C07284=1031.312,-76.674,415.942,167.658,41.793,157.756
C07285=1031.305,-76.924,415.953,167.656,41.794,157.756
C07286=1031.300,-77.174,415.964,167.653,41.796,157.756
C07287=1031.294,-77.423,415.975,167.650,41.797,157.756
C07288=1031.287,-77.673,415.985,167.647,41.798,157.757
C07289=1031.281,-77.922,415.996,167.644,41.799,157.757
C07290=1031.275,-78.172,416.007,167.642,41.801,157.757
C07291=1031.269,-78.422,416.018,167.639,41.802,157.757
C07292=1031.263,-78.672,416.029,167.636,41.803,157.757
C07293=1031.258,-78.921,416.040,167.633,41.805,157.757
C07294=1031.251,-79.171,416.051,167.630,41.806,157.757
C07295=1031.246,-79.421,416.062,167.628,41.808,157.757
C07296=1031.239,-79.670,416.073,167.625,41.809,157.757
C07297=1031.233,-79.920,416.084,167.622,41.811,157.757
C07298=1031.227,-80.170,416.094,167.619,41.812,157.757
C07299=1031.222,-80.420,416.105,167.617,41.814,157.757
C07300=1031.214,-80.670,416.116,167.614,41.815,157.757
C07301=1031.209,-80.919,416.126,167.611,41.816,157.757
C07302=1031.202,-81.168,416.137,167.608,41.818,157.758
C07303=1031.196,-81.418,416.148,167.606,41.820,157.758
C07304=1031.190,-81.669,416.158,167.603,41.821,157.758
C07305=1031.184,-81.918,416.168,167.600,41.823,157.758
C07306=1031.178,-82.167,416.179,167.597,41.825,157.758
C07307=1031.171,-82.417,416.190,167.594,41.826,157.758
C07308=1031.165,-82.667,416.201,167.592,41.827,157.758
C07309=1031.160,-82.917,416.211,167.589,41.828,157.758
C07310=1031.153,-83.166,416.221,167.586,41.830,157.758
C07311=1031.147,-83.416,416.233,167.582,41.832,157.758
C07312=1031.141,-83.666,416.243,167.580,41.833,157.758
C07313=1031.135,-83.915,416.253,167.577,41.835,157.759
C07314=1031.128,-84.199,416.266,167.574,41.837,157.759
C07315=1031.121,-84.485,416.278,167.570,41.839,157.759
C07316=1031.114,-84.769,416.290,167.568,41.840,157.759
C07317=1031.107,-85.054,416.302,167.564,41.842,157.759
C07318=1031.101,-85.303,416.312,167.561,41.843,157.759
C07319=1031.096,-85.553,416.322,167.558,41.845,157.759
C07320=1031.089,-85.803,416.333,167.556,41.847,157.759
C07321=1031.083,-86.053,416.344,167.553,41.848,157.759
C07322=1031.077,-86.303,416.354,167.550,41.850,157.760
C07323=1031.071,-86.552,416.364,167.547,41.851,157.760
C07324=1031.065,-86.802,416.374,167.545,41.852,157.760
C07325=1031.059,-87.051,416.385,167.542,41.854,157.760
C07326=1031.053,-87.302,416.396,167.539,41.855,157.760
C07327=1031.046,-87.551,416.405,167.536,41.857,157.760
C07328=1031.041,-87.801,416.416,167.534,41.859,157.760
C07329=1031.035,-88.050,416.427,167.531,41.860,157.760
C07330=1031.029,-88.300,416.437,167.528,41.862,157.760
C07331=1031.023,-88.550,416.448,167.525,41.863,157.760
C07332=1031.017,-88.799,416.457,167.522,41.865,157.760
C07333=1031.010,-89.050,416.468,167.520,41.866,157.761
C07334=1031.004,-89.299,416.478,167.517,41.868,157.761
C07335=1030.999,-89.549,416.489,167.514,41.869,157.761
C07336=1030.992,-89.798,416.499,167.510,41.871,157.761
C07337=1030.987,-90.048,416.509,167.508,41.873,157.761
C07338=1030.981,-90.298,416.520,167.505,41.874,157.761
C07339=1030.975,-90.547,416.530,167.502,41.876,157.761
C07340=1030.969,-90.797,416.541,167.499,41.877,157.761
C07341=1030.963,-91.047,416.550,167.496,41.878,157.761
C07342=1030.957,-91.296,416.561,167.494,41.880,157.761
C07343=1030.951,-91.546,416.571,167.491,41.882,157.761
C07344=1030.945,-91.796,416.582,167.488,41.883,157.761
C07345=1030.938,-92.046,416.591,167.485,41.885,157.762
C07346=1030.933,-92.296,416.602,167.483,41.887,157.762
C07347=1030.926,-92.545,416.612,167.480,41.888,157.762
C07348=1030.921,-92.795,416.622,167.477,41.889,157.762
C07349=1030.915,-93.045,416.632,167.475,41.891,157.762
C07350=1030.909,-93.295,416.643,167.472,41.892,157.762
C07351=1030.903,-93.544,416.653,167.469,41.894,157.762
C07352=1030.897,-93.794,416.663,167.466,41.895,157.762
C07353=1030.892,-94.044,416.673,167.463,41.897,157.762
C07354=1030.885,-94.293,416.683,167.460,41.899,157.762
C07355=1030.880,-94.543,416.694,167.457,41.900,157.762
C07356=1030.873,-94.793,416.704,167.454,41.902,157.763
C07357=1030.868,-95.043,416.714,167.451,41.903,157.763
C07358=1030.862,-95.292,416.724,167.448,41.904,157.763
C07359=1030.856,-95.542,416.734,167.446,41.906,157.763
C07360=1030.850,-95.792,416.744,167.443,41.908,157.763
C07361=1030.844,-96.042,416.754,167.440,41.909,157.763
C07362=1030.839,-96.290,416.764,167.437,41.911,157.763
C07363=1030.833,-96.540,416.774,167.435,41.913,157.763
C07364=1030.827,-96.790,416.784,167.432,41.914,157.763
C07365=1030.821,-97.040,416.795,167.429,41.915,157.763
C07366=1030.815,-97.290,416.804,167.426,41.917,157.764
C07367=1030.810,-97.540,416.814,167.424,41.918,157.764
C07368=1030.803,-97.789,416.824,167.421,41.920,157.764
C07369=1030.797,-98.039,416.834,167.417,41.922,157.764
C07370=1030.792,-98.289,416.844,167.414,41.924,157.764
C07371=1030.785,-98.539,416.854,167.412,41.925,157.764
C07372=1030.779,-98.788,416.864,167.409,41.927,157.764
C07373=1030.773,-99.038,416.873,167.406,41.929,157.764
C07374=1030.768,-99.288,416.883,167.404,41.930,157.764
C07375=1030.761,-99.538,416.893,167.401,41.932,157.764
C07376=1030.755,-99.787,416.903,167.398,41.934,157.765
C07377=1030.749,-100.037,416.913,167.394,41.936,157.765
C07378=1030.743,-100.324,416.924,167.392,41.937,157.765
C07379=1030.736,-100.611,416.935,167.388,41.939,157.765
C07380=1030.729,-100.898,416.946,167.385,41.941,157.765
C07381=1030.722,-101.184,416.957,167.382,41.943,157.765
C07382=1030.716,-101.434,416.967,167.379,41.945,157.765
C07383=1030.710,-101.684,416.977,167.376,41.946,157.765
C07384=1030.704,-101.934,416.986,167.373,41.948,157.766
C07385=1030.698,-102.184,416.996,167.371,41.950,157.766
C07386=1030.693,-102.433,417.005,167.367,41.952,157.766
C07387=1030.686,-102.683,417.015,167.364,41.954,157.766
C07388=1030.681,-102.933,417.025,167.361,41.955,157.766
C07389=1030.674,-103.182,417.035,167.359,41.956,157.766
C07390=1030.668,-103.432,417.045,167.356,41.958,157.766
C07391=1030.662,-103.682,417.054,167.353,41.960,157.766
C07392=1030.657,-103.931,417.063,167.351,41.962,157.766
C07393=1030.651,-104.182,417.073,167.348,41.964,157.767
C07394=1030.645,-104.431,417.083,167.344,41.965,157.767
C07395=1030.639,-104.681,417.092,167.341,41.967,157.767
C07396=1030.633,-104.931,417.102,167.339,41.968,157.767
C07397=1030.627,-105.180,417.111,167.336,41.970,157.767
C07398=1030.622,-105.430,417.121,167.333,41.972,157.767
C07399=1030.616,-105.680,417.131,167.330,41.974,157.767
C07400=1030.610,-105.930,417.140,167.328,41.975,157.767
C07401=1030.603,-106.180,417.150,167.325,41.977,157.767
C07402=1030.598,-106.429,417.159,167.321,41.979,157.768
C07403=1030.592,-106.678,417.169,167.319,41.981,157.768
C07404=1030.586,-106.929,417.179,167.316,41.983,157.768
C07405=1030.580,-107.179,417.188,167.313,41.984,157.768
C07406=1030.575,-107.428,417.197,167.310,41.985,157.768
C07407=1030.569,-107.678,417.206,167.308,41.987,157.768
C07408=1030.562,-107.928,417.216,167.305,41.989,157.768
C07409=1030.556,-108.177,417.225,167.301,41.991,157.768
C07410=1030.551,-108.427,417.235,167.299,41.993,157.768
C07411=1030.545,-108.677,417.244,167.296,41.995,157.769
C07412=1030.539,-108.927,417.253,167.293,41.996,157.769
C07413=1030.533,-109.176,417.262,167.290,41.998,157.769
C07414=1030.527,-109.426,417.272,167.288,42.000,157.769
C07415=1030.521,-109.676,417.281,167.284,42.002,157.769
C07416=1030.515,-109.926,417.290,167.281,42.004,157.769
C07417=1030.509,-110.175,417.300,167.279,42.005,157.769
C07418=1030.503,-110.425,417.309,167.276,42.008,157.770
C07419=1030.497,-110.675,417.318,167.273,42.010,157.770
C07420=1030.492,-110.924,417.327,167.270,42.011,157.770
C07421=1030.486,-111.174,417.337,167.267,42.013,157.770
C07422=1030.480,-111.425,417.346,167.264,42.015,157.770
C07423=1030.474,-111.674,417.355,167.262,42.017,157.770
C07424=1030.468,-111.923,417.364,167.259,42.019,157.770
C07425=1030.462,-112.174,417.373,167.256,42.020,157.770
C07426=1030.457,-112.423,417.382,167.252,42.022,157.771
C07427=1030.450,-112.673,417.392,167.250,42.024,157.771
C07428=1030.444,-112.923,417.401,167.247,42.026,157.771
C07429=1030.439,-113.172,417.410,167.244,42.028,157.771
C07430=1030.433,-113.422,417.420,167.242,42.029,157.771
C07431=1030.427,-113.672,417.428,167.239,42.031,157.771
C07432=1030.421,-113.922,417.438,167.235,42.033,157.771
C07433=1030.415,-114.172,417.446,167.233,42.035,157.771
C07434=1030.410,-114.421,417.456,167.230,42.037,157.772
C07435=1030.404,-114.671,417.465,167.227,42.038,157.772
C07436=1030.398,-114.920,417.473,167.224,42.040,157.772
C07437=1030.392,-115.170,417.483,167.222,42.042,157.772
C07438=1030.386,-115.420,417.492,167.218,42.044,157.772
C07439=1030.380,-115.670,417.501,167.215,42.046,157.772
C07440=1030.374,-115.920,417.510,167.213,42.047,157.772
C07441=1030.369,-116.169,417.519,167.210,42.050,157.772
C07442=1030.361,-116.456,417.528,167.206,42.052,157.773
C07443=1030.355,-116.743,417.539,167.203,42.054,157.773
C07444=1030.348,-117.028,417.549,167.200,42.056,157.773
C07445=1030.342,-117.315,417.559,167.196,42.058,157.773
C07446=1030.336,-117.565,417.568,167.194,42.060,157.773
C07447=1030.330,-117.815,417.577,167.191,42.062,157.773
C07448=1030.325,-118.064,417.587,167.188,42.064,157.774
C07449=1030.318,-118.314,417.595,167.185,42.066,157.774
C07450=1030.312,-118.563,417.604,167.182,42.068,157.774
C07451=1030.306,-118.814,417.613,167.179,42.070,157.774
C07452=1030.301,-119.064,417.622,167.177,42.071,157.774
C07453=1030.294,-119.313,417.630,167.174,42.073,157.774
C07454=1030.288,-119.563,417.639,167.170,42.075,157.774
C07455=1030.283,-119.813,417.648,167.168,42.078,157.774
C07456=1030.277,-120.063,417.657,167.165,42.079,157.775
C07457=1030.272,-120.313,417.666,167.162,42.081,157.775
C07458=1030.265,-120.561,417.674,167.159,42.083,157.775
C07459=1030.260,-120.812,417.683,167.156,42.085,157.775
C07460=1030.254,-121.061,417.692,167.153,42.087,157.775
C07461=1030.248,-121.312,417.700,167.151,42.089,157.775
C07462=1030.242,-121.561,417.709,167.148,42.091,157.775
C07463=1030.236,-121.811,417.718,167.144,42.093,157.776
C07464=1030.231,-122.061,417.726,167.142,42.095,157.776
C07465=1030.225,-122.311,417.736,167.139,42.096,157.776
C07466=1030.219,-122.560,417.744,167.136,42.099,157.776
C07467=1030.213,-122.810,417.753,167.134,42.101,157.776
C07468=1030.208,-123.060,417.761,167.130,42.103,157.776
C07469=1030.202,-123.309,417.770,167.127,42.104,157.776
C07470=1030.196,-123.559,417.779,167.124,42.106,157.777
C07471=1030.190,-123.809,417.787,167.122,42.108,157.777
C07472=1030.184,-124.059,417.796,167.119,42.110,157.777
C07473=1030.179,-124.309,417.804,167.116,42.112,157.777
C07474=1030.173,-124.558,417.813,167.113,42.114,157.777
C07475=1030.167,-124.808,417.822,167.110,42.116,157.777
C07476=1030.161,-125.058,417.830,167.108,42.118,157.777
C07477=1030.155,-125.308,417.839,167.104,42.120,157.778
C07478=1030.150,-125.558,417.847,167.101,42.122,157.778
C07479=1030.144,-125.807,417.855,167.098,42.124,157.778
C07480=1030.138,-126.058,417.864,167.096,42.126,157.778
C07481=1030.132,-126.307,417.872,167.092,42.128,157.778
C07482=1030.126,-126.556,417.881,167.090,42.130,157.778
C07483=1030.121,-126.807,417.890,167.087,42.133,157.779
C07484=1030.115,-127.056,417.898,167.084,42.134,157.779
C07485=1030.109,-127.306,417.907,167.082,42.136,157.779
C07486=1030.103,-127.556,417.914,167.078,42.139,157.779
C07487=1030.097,-127.806,417.923,167.075,42.140,157.779
C07488=1030.092,-128.055,417.932,167.073,42.142,157.779
C07489=1030.087,-128.305,417.941,167.070,42.143,157.779
C07490=1030.082,-128.554,417.951,167.067,42.144,157.779
C07491=1030.080,-128.803,417.962,167.065,42.145,157.779
C07492=1030.076,-129.053,417.973,167.063,42.144,157.779
C07493=1030.074,-129.303,417.984,167.059,42.144,157.779
C07494=1030.072,-129.554,417.996,167.058,42.143,157.778
C07495=1030.071,-129.803,418.009,167.056,42.142,157.778
C07496=1030.071,-130.053,418.022,167.053,42.139,157.777
C07497=1030.071,-130.303,418.036,167.051,42.137,157.777
C07498=1030.071,-130.553,418.050,167.049,42.134,157.776
C07499=1030.073,-130.803,418.066,167.048,42.131,157.776
C07500=1030.075,-131.053,418.082,167.045,42.127,157.775
C07501=1030.077,-131.302,418.098,167.044,42.123,157.774
C07502=1030.081,-131.553,418.115,167.043,42.118,157.773
C07503=1030.085,-131.803,418.132,167.042,42.112,157.772
C07504=1030.089,-132.053,418.150,167.040,42.107,157.771
C07505=1030.095,-132.302,418.169,167.039,42.101,157.770
C07506=1029.776,-132.327,417.864,166.990,42.343,157.807
C07507=1029.771,-132.078,417.846,166.992,42.349,157.808
C07508=1029.767,-131.828,417.828,166.993,42.355,157.809
C07509=1029.762,-131.577,417.810,166.994,42.360,157.811
C07510=1029.759,-131.327,417.794,166.996,42.365,157.811
C07511=1029.756,-131.077,417.777,166.997,42.369,157.812
C07512=1029.755,-130.827,417.762,166.999,42.373,157.813
C07513=1029.753,-130.578,417.747,167.001,42.376,157.814
C07514=1029.752,-130.328,417.732,167.003,42.379,157.814
C07515=1029.752,-130.078,417.718,167.004,42.382,157.815
C07516=1029.753,-129.828,417.705,167.007,42.383,157.815
C07517=1029.754,-129.578,417.692,167.009,42.385,157.816
C07518=1029.755,-129.328,417.680,167.011,42.386,157.816
C07519=1029.758,-129.079,417.668,167.013,42.387,157.816
C07520=1029.760,-128.829,417.657,167.016,42.386,157.816
C07521=1029.764,-128.579,417.646,167.018,42.386,157.816
C07522=1029.769,-128.330,417.636,167.021,42.386,157.817
C07523=1029.773,-128.080,417.627,167.024,42.384,157.816
C07524=1029.778,-127.830,417.619,167.027,42.382,157.816
C07525=1029.784,-127.580,417.610,167.029,42.380,157.816
C07526=1029.790,-127.332,417.602,167.032,42.378,157.816
C07527=1029.795,-127.082,417.593,167.036,42.376,157.816
C07528=1029.802,-126.832,417.585,167.038,42.374,157.816
C07529=1029.807,-126.582,417.576,167.041,42.372,157.816
C07530=1029.812,-126.332,417.568,167.044,42.370,157.816
C07531=1029.819,-126.082,417.560,167.047,42.368,157.815
C07532=1029.824,-125.833,417.551,167.050,42.366,157.815
C07533=1029.830,-125.583,417.543,167.053,42.364,157.815
C07534=1029.836,-125.333,417.534,167.055,42.362,157.815
C07535=1029.841,-125.083,417.526,167.059,42.360,157.815
C07536=1029.848,-124.833,417.518,167.062,42.358,157.815
C07537=1029.854,-124.584,417.508,167.064,42.355,157.814
C07538=1029.860,-124.334,417.501,167.068,42.353,157.814
C07539=1029.865,-124.084,417.492,167.070,42.352,157.814
C07540=1029.871,-123.834,417.483,167.073,42.349,157.814
C07541=1029.877,-123.584,417.474,167.076,42.347,157.814
C07542=1029.883,-123.335,417.466,167.078,42.345,157.814
C07543=1029.888,-123.085,417.457,167.082,42.344,157.814
C07544=1029.894,-122.835,417.448,167.085,42.342,157.813
C07545=1029.900,-122.586,417.441,167.087,42.339,157.813
C07546=1029.906,-122.335,417.432,167.090,42.337,157.813
C07547=1029.911,-122.086,417.422,167.094,42.335,157.813
C07548=1029.917,-121.836,417.414,167.096,42.334,157.813
C07549=1029.923,-121.586,417.406,167.099,42.331,157.813
C07550=1029.929,-121.337,417.397,167.102,42.329,157.813
C07551=1029.935,-121.087,417.388,167.105,42.327,157.812
C07552=1029.940,-120.837,417.379,167.108,42.326,157.812
C07553=1029.947,-120.587,417.371,167.110,42.323,157.812
C07554=1029.952,-120.338,417.362,167.113,42.321,157.812
C07555=1029.958,-120.087,417.353,167.116,42.320,157.812
C07556=1029.963,-119.838,417.344,167.120,42.318,157.812
C07557=1029.970,-119.588,417.335,167.122,42.316,157.812
C07558=1029.976,-119.338,417.327,167.125,42.313,157.811
C07559=1029.981,-119.088,417.318,167.127,42.311,157.811
C07560=1029.987,-118.839,417.309,167.131,42.310,157.811
C07561=1029.993,-118.589,417.300,167.134,42.308,157.811
C07562=1029.998,-118.339,417.291,167.137,42.306,157.811
C07563=1030.005,-118.089,417.283,167.139,42.303,157.811
C07564=1030.010,-117.840,417.274,167.143,42.302,157.811
C07565=1030.016,-117.590,417.265,167.145,42.300,157.810
C07566=1030.022,-117.340,417.256,167.148,42.298,157.810
C07567=1030.029,-117.054,417.246,167.152,42.295,157.810
C07568=1030.035,-116.768,417.235,167.154,42.293,157.810
C07569=1030.042,-116.481,417.226,167.158,42.292,157.810
C07570=1030.049,-116.195,417.215,167.162,42.289,157.810
C07571=1030.055,-115.945,417.206,167.164,42.287,157.810
C07572=1030.061,-115.695,417.197,167.167,42.285,157.809
C07573=1030.066,-115.446,417.188,167.170,42.284,157.809
C07574=1030.073,-115.196,417.179,167.173,42.281,157.809
C07575=1030.078,-114.947,417.170,167.176,42.279,157.809
C07576=1030.084,-114.696,417.161,167.179,42.277,157.809
C07577=1030.090,-114.446,417.152,167.181,42.275,157.809
C07578=1030.096,-114.197,417.143,167.185,42.274,157.809
C07579=1030.102,-113.947,417.134,167.188,42.272,157.809
C07580=1030.107,-113.697,417.125,167.190,42.270,157.808
C07581=1030.113,-113.447,417.116,167.193,42.268,157.808
C07582=1030.119,-113.198,417.106,167.196,42.266,157.808
C07583=1030.125,-112.948,417.098,167.199,42.265,157.808
C07584=1030.131,-112.698,417.088,167.202,42.263,157.808
C07585=1030.136,-112.448,417.080,167.205,42.260,157.808
C07586=1030.142,-112.199,417.070,167.207,42.258,157.808
C07587=1030.148,-111.949,417.060,167.210,42.257,157.807
C07588=1030.154,-111.699,417.052,167.213,42.255,157.807
C07589=1030.160,-111.449,417.042,167.217,42.253,157.807
C07590=1030.166,-111.199,417.033,167.219,42.251,157.807
C07591=1030.171,-110.950,417.024,167.222,42.249,157.807
C07592=1030.177,-110.700,417.015,167.225,42.247,157.807
C07593=1030.184,-110.450,417.005,167.227,42.246,157.807
C07594=1030.189,-110.200,416.997,167.231,42.244,157.807
C07595=1030.195,-109.951,416.987,167.234,42.242,157.807
C07596=1030.201,-109.701,416.978,167.236,42.240,157.806
C07597=1030.207,-109.452,416.968,167.239,42.238,157.806
C07598=1030.213,-109.201,416.959,167.242,42.237,157.806
C07599=1030.219,-108.951,416.950,167.246,42.235,157.806
C07600=1030.224,-108.702,416.941,167.248,42.233,157.806
C07601=1030.231,-108.453,416.931,167.251,42.230,157.806
C07602=1030.236,-108.202,416.922,167.253,42.229,157.806
C07603=1030.243,-107.952,416.913,167.256,42.227,157.805
C07604=1030.248,-107.703,416.904,167.260,42.225,157.805
C07605=1030.254,-107.453,416.894,167.263,42.223,157.805
C07606=1030.261,-107.204,416.884,167.265,42.221,157.805
C07607=1030.266,-106.953,416.876,167.268,42.219,157.805
C07608=1030.272,-106.704,416.866,167.271,42.218,157.805
C07609=1030.278,-106.454,416.857,167.273,42.216,157.805
C07610=1030.284,-106.204,416.847,167.277,42.214,157.805
C07611=1030.290,-105.954,416.837,167.280,42.213,157.805
C07612=1030.295,-105.705,416.828,167.283,42.211,157.804
C07613=1030.302,-105.456,416.818,167.285,42.209,157.804
C07614=1030.308,-105.206,416.809,167.288,42.207,157.804
C07615=1030.314,-104.956,416.799,167.291,42.206,157.804
C07616=1030.319,-104.705,416.790,167.294,42.204,157.804
C07617=1030.325,-104.456,416.780,167.297,42.202,157.804
C07618=1030.331,-104.206,416.771,167.300,42.200,157.804
C07619=1030.337,-103.957,416.761,167.302,42.198,157.804
C07620=1030.343,-103.707,416.752,167.305,42.197,157.803
C07621=1030.348,-103.457,416.742,167.308,42.195,157.803
C07622=1030.354,-103.208,416.732,167.311,42.193,157.803
C07623=1030.360,-102.958,416.723,167.314,42.191,157.803
C07624=1030.366,-102.708,416.713,167.317,42.189,157.803
C07625=1030.373,-102.458,416.704,167.320,42.188,157.803
C07626=1030.378,-102.208,416.694,167.323,42.186,157.803
C07627=1030.384,-101.959,416.684,167.325,42.185,157.803
C07628=1030.390,-101.709,416.675,167.328,42.183,157.803
C07629=1030.396,-101.459,416.665,167.332,42.181,157.803
C07630=1030.402,-101.210,416.654,167.334,42.179,157.802
C07631=1030.408,-100.923,416.643,167.337,42.177,157.802
C07632=1030.416,-100.636,416.632,167.341,42.175,157.802
C07633=1030.422,-100.349,416.621,167.344,42.173,157.802
C07634=1030.429,-100.063,416.610,167.347,42.171,157.802
C07635=1030.435,-99.813,416.601,167.350,42.169,157.802
C07636=1030.441,-99.563,416.591,167.352,42.167,157.802
C07637=1030.447,-99.313,416.581,167.356,42.165,157.802
C07638=1030.453,-99.063,416.572,167.359,42.164,157.802
C07639=1030.460,-98.814,416.561,167.362,42.163,157.801
C07640=1030.465,-98.564,416.551,167.364,42.161,157.801
C07641=1030.471,-98.314,416.542,167.367,42.159,157.801
C07642=1030.477,-98.064,416.532,167.370,42.157,157.801
C07643=1030.483,-97.815,416.522,167.373,42.155,157.801
C07644=1030.489,-97.564,416.512,167.376,42.154,157.801
C07645=1030.495,-97.315,416.502,167.379,42.152,157.801
C07646=1030.501,-97.065,416.492,167.382,42.151,157.801
C07647=1030.506,-96.816,416.483,167.384,42.149,157.800
C07648=1030.512,-96.566,416.473,167.387,42.147,157.800
C07649=1030.518,-96.317,416.462,167.390,42.146,157.800
C07650=1030.524,-96.067,416.452,167.393,42.144,157.800
C07651=1030.530,-95.817,416.443,167.395,42.142,157.800
C07652=1030.536,-95.567,416.432,167.398,42.141,157.800
C07653=1030.542,-95.318,416.422,167.401,42.140,157.800
C07654=1030.547,-95.067,416.412,167.405,42.138,157.800
C07655=1030.554,-94.818,416.402,167.407,42.136,157.800
C07656=1030.559,-94.568,416.391,167.410,42.134,157.800
C07657=1030.565,-94.318,416.382,167.413,42.133,157.800
C07658=1030.571,-94.069,416.371,167.416,42.131,157.799
C07659=1030.577,-93.819,416.361,167.418,42.129,157.799
C07660=1030.583,-93.570,416.351,167.421,42.128,157.799
C07661=1030.589,-93.320,416.341,167.424,42.127,157.799
C07662=1030.595,-93.070,416.331,167.427,42.125,157.799
C07663=1030.601,-92.821,416.321,167.429,42.123,157.799
C07664=1030.607,-92.570,416.310,167.432,42.122,157.799
C07665=1030.612,-92.321,416.300,167.436,42.120,157.799
C07666=1030.618,-92.071,416.290,167.439,42.118,157.799
C07667=1030.624,-91.822,416.279,167.441,42.117,157.799
C07668=1030.630,-91.572,416.270,167.444,42.115,157.799
C07669=1030.636,-91.322,416.259,167.447,42.113,157.798
C07670=1030.642,-91.073,416.249,167.449,42.112,157.798
C07671=1030.648,-90.822,416.239,167.452,42.111,157.798
C07672=1030.654,-90.573,416.229,167.455,42.109,157.798
C07673=1030.660,-90.322,416.218,167.458,42.107,157.798
C07674=1030.667,-90.073,416.208,167.461,42.106,157.798
C07675=1030.672,-89.823,416.198,167.463,42.104,157.798
C07676=1030.679,-89.574,416.187,167.466,42.102,157.798
C07677=1030.684,-89.324,416.176,167.470,42.100,157.798
C07678=1030.690,-89.074,416.166,167.473,42.099,157.798
C07679=1030.696,-88.825,416.156,167.475,42.098,157.798
C07680=1030.702,-88.575,416.146,167.478,42.096,157.797
C07681=1030.708,-88.326,416.136,167.481,42.095,157.797
C07682=1030.714,-88.076,416.125,167.484,42.093,157.797
C07683=1030.721,-87.826,416.115,167.486,42.091,157.797
C07684=1030.726,-87.576,416.104,167.489,42.089,157.797
C07685=1030.732,-87.326,416.094,167.492,42.088,157.797
C07686=1030.738,-87.077,416.083,167.495,42.087,157.797
C07687=1030.744,-86.827,416.073,167.497,42.085,157.797
C07688=1030.750,-86.578,416.063,167.500,42.084,157.797
C07689=1030.757,-86.328,416.052,167.503,42.082,157.797
C07690=1030.763,-86.078,416.042,167.507,42.080,157.797
C07691=1030.768,-85.828,416.031,167.509,42.079,157.797
C07692=1030.774,-85.579,416.020,167.512,42.077,157.796
C07693=1030.780,-85.329,416.011,167.515,42.075,157.796
C07694=1030.786,-85.080,416.000,167.517,42.074,157.796
C07695=1030.793,-84.794,415.988,167.520,42.072,157.796
C07696=1030.801,-84.510,415.976,167.524,42.070,157.796
C07697=1030.808,-84.225,415.964,167.527,42.069,157.796
C07698=1030.814,-83.941,415.953,167.530,42.067,157.796
C07699=1030.820,-83.691,415.942,167.533,42.065,157.796
C07700=1030.827,-83.442,415.931,167.536,42.063,157.796
C07701=1030.833,-83.192,415.920,167.539,42.062,157.795
C07702=1030.838,-82.942,415.910,167.541,42.060,157.795
C07703=1030.845,-82.692,415.900,167.544,42.059,157.795
C07704=1030.851,-82.443,415.889,167.547,42.057,157.795
C07705=1030.858,-82.193,415.878,167.550,42.056,157.795
C07706=1030.863,-81.943,415.868,167.552,42.054,157.795
C07707=1030.869,-81.694,415.857,167.556,42.052,157.795
C07708=1030.876,-81.444,415.846,167.559,42.050,157.795
C07709=1030.882,-81.194,415.836,167.562,42.049,157.795
C07710=1030.888,-80.945,415.825,167.564,42.047,157.795
C07711=1030.894,-80.695,415.815,167.567,42.046,157.794
C07712=1030.900,-80.445,415.804,167.570,42.045,157.794
C07713=1030.906,-80.195,415.794,167.573,42.043,157.794
C07714=1030.912,-79.946,415.783,167.575,42.041,157.794
C07715=1030.918,-79.696,415.771,167.578,42.040,157.794
C07716=1030.924,-79.446,415.761,167.581,42.038,157.794
C07717=1030.931,-79.197,415.750,167.584,42.037,157.794
C07718=1030.937,-78.947,415.739,167.586,42.035,157.794
C07719=1030.943,-78.697,415.728,167.589,42.034,157.794
C07720=1030.948,-78.448,415.717,167.592,42.032,157.794
C07721=1030.955,-78.198,415.706,167.595,42.031,157.794
C07722=1030.961,-77.948,415.695,167.598,42.030,157.794
C07723=1030.966,-77.699,415.684,167.600,42.028,157.793
C07724=1030.973,-77.449,415.673,167.603,42.027,157.793
C07725=1030.979,-77.199,415.663,167.606,42.025,157.793
C07726=1030.985,-76.950,415.652,167.609,42.024,157.793
C07727=1030.991,-76.700,415.641,167.611,42.022,157.793
C07728=1030.997,-76.450,415.630,167.614,42.021,157.793
C07729=1031.003,-76.201,415.619,167.617,42.019,157.793
C07730=1031.009,-75.951,415.608,167.620,42.018,157.793
C07731=1031.015,-75.701,415.597,167.623,42.016,157.793
C07732=1031.020,-75.452,415.586,167.625,42.015,157.793
C07733=1031.028,-75.202,415.575,167.628,42.014,157.793
C07734=1031.033,-74.952,415.564,167.631,42.012,157.793
C07735=1031.040,-74.702,415.553,167.634,42.011,157.793
C07736=1031.045,-74.453,415.542,167.637,42.010,157.793
C07737=1031.051,-74.203,415.531,167.639,42.008,157.792
C07738=1031.058,-73.953,415.519,167.642,42.007,157.792
C07739=1031.064,-73.704,415.509,167.645,42.005,157.792
C07740=1031.070,-73.454,415.497,167.648,42.004,157.792
C07741=1031.075,-73.204,415.486,167.651,42.003,157.792
C07742=1031.081,-72.955,415.475,167.653,42.001,157.792
C07743=1031.087,-72.705,415.463,167.656,42.000,157.792
C07744=1031.093,-72.455,415.452,167.659,41.999,157.792
C07745=1031.099,-72.205,415.441,167.662,41.997,157.792
C07746=1031.105,-71.956,415.430,167.665,41.996,157.792
C07747=1031.110,-71.707,415.418,167.668,41.995,157.792
C07748=1031.117,-71.456,415.407,167.670,41.993,157.792
C07749=1031.122,-71.207,415.396,167.672,41.992,157.792
C07750=1031.129,-70.957,415.384,167.675,41.991,157.792
C07751=1031.135,-70.708,415.373,167.678,41.989,157.792
C07752=1031.141,-70.458,415.362,167.681,41.988,157.792
C07753=1031.146,-70.208,415.349,167.683,41.987,157.792
C07754=1031.153,-69.958,415.338,167.686,41.985,157.791
C07755=1031.159,-69.709,415.327,167.689,41.984,157.791
C07756=1031.165,-69.460,415.316,167.692,41.983,157.791
C07757=1031.171,-69.210,415.304,167.695,41.981,157.791
C07758=1031.176,-68.960,415.293,167.697,41.980,157.791
C07759=1031.183,-68.678,415.281,167.700,41.979,157.791
C07760=1031.190,-68.395,415.268,167.703,41.978,157.791
C07761=1031.197,-68.113,415.254,167.707,41.976,157.791
C07762=1031.204,-67.830,415.241,167.710,41.975,157.791
C07763=1031.210,-67.580,415.230,167.712,41.973,157.791
C07764=1031.216,-67.330,415.219,167.715,41.972,157.791
C07765=1031.222,-67.081,415.206,167.718,41.971,157.791
C07766=1031.228,-66.831,415.195,167.721,41.969,157.791
C07767=1031.234,-66.582,415.183,167.724,41.968,157.791
C07768=1031.240,-66.332,415.172,167.726,41.967,157.791
C07769=1031.247,-66.082,415.161,167.729,41.965,157.791
C07770=1031.252,-65.833,415.149,167.732,41.964,157.791
C07771=1031.258,-65.583,415.137,167.734,41.963,157.791
C07772=1031.265,-65.333,415.126,167.737,41.961,157.790
C07773=1031.271,-65.084,415.114,167.739,41.960,157.790
C07774=1031.277,-64.834,415.103,167.742,41.959,157.790
C07775=1031.282,-64.585,415.091,167.745,41.957,157.790
C07776=1031.289,-64.334,415.080,167.748,41.956,157.790
C07777=1031.295,-64.086,415.068,167.751,41.954,157.790
C07778=1031.301,-63.835,415.057,167.753,41.953,157.790
C07779=1031.307,-63.586,415.044,167.756,41.952,157.790
C07780=1031.313,-63.336,415.033,167.759,41.950,157.790
C07781=1031.319,-63.086,415.021,167.762,41.949,157.790
C07782=1031.326,-62.836,415.010,167.765,41.948,157.790
C07783=1031.331,-62.587,414.998,167.766,41.947,157.790
C07784=1031.338,-62.338,414.986,167.769,41.946,157.790
C07785=1031.343,-62.088,414.975,167.772,41.944,157.790
C07786=1031.350,-61.838,414.963,167.775,41.943,157.790
C07787=1031.356,-61.588,414.952,167.778,41.942,157.790
C07788=1031.362,-61.339,414.940,167.781,41.941,157.790
C07789=1031.368,-61.090,414.928,167.783,41.939,157.789
C07790=1031.375,-60.839,414.917,167.786,41.938,157.789
C07791=1031.381,-60.590,414.905,167.789,41.936,157.789
C07792=1031.387,-60.341,414.892,167.792,41.935,157.789
C07793=1031.393,-60.090,414.881,167.795,41.934,157.789
C07794=1031.399,-59.842,414.870,167.797,41.932,157.789
C07795=1031.406,-59.592,414.858,167.799,41.931,157.789
C07796=1031.411,-59.341,414.846,167.802,41.930,157.789
C07797=1031.418,-59.092,414.834,167.805,41.928,157.789
C07798=1031.424,-58.843,414.822,167.808,41.927,157.789
C07799=1031.430,-58.593,414.811,167.811,41.926,157.789
C07800=1031.436,-58.343,414.798,167.813,41.924,157.789
C07801=1031.443,-58.093,414.786,167.816,41.923,157.789
C07802=1031.449,-57.844,414.775,167.819,41.922,157.789
C07803=1031.455,-57.594,414.763,167.822,41.920,157.789
C07804=1031.461,-57.344,414.751,167.825,41.919,157.789
C07805=1031.468,-57.095,414.739,167.827,41.918,157.788
C07806=1031.474,-56.846,414.727,167.829,41.917,157.788
C07807=1031.480,-56.595,414.716,167.832,41.915,157.788
C07808=1031.486,-56.346,414.704,167.835,41.914,157.788
C07809=1031.493,-56.096,414.692,167.838,41.913,157.788
C07810=1031.499,-55.847,414.680,167.840,41.912,157.788
C07811=1031.505,-55.598,414.668,167.843,41.910,157.788
C07812=1031.511,-55.347,414.656,167.846,41.909,157.788
C07813=1031.518,-55.098,414.644,167.849,41.907,157.788
C07814=1031.524,-54.848,414.632,167.852,41.906,157.788
C07815=1031.530,-54.599,414.620,167.854,41.905,157.788
C07816=1031.536,-54.349,414.608,167.856,41.903,157.788
C07817=1031.543,-54.100,414.596,167.859,41.902,157.788
C07818=1031.549,-53.849,414.584,167.862,41.901,157.788
C07819=1031.555,-53.600,414.573,167.865,41.899,157.787
C07820=1031.562,-53.350,414.561,167.867,41.898,157.787
C07821=1031.567,-53.101,414.548,167.870,41.896,157.787
C07822=1031.574,-52.852,414.536,167.873,41.895,157.787
C07823=1031.581,-52.569,414.523,167.876,41.894,157.787
C07824=1031.588,-52.289,414.509,167.879,41.893,157.787
C07825=1031.595,-52.007,414.496,167.882,41.891,157.787
C07826=1031.603,-51.727,414.482,167.885,41.890,157.787
C07827=1031.609,-51.477,414.469,167.888,41.888,157.787
C07828=1031.615,-51.227,414.458,167.891,41.887,157.787
C07829=1031.622,-50.978,414.446,167.894,41.886,157.787
C07830=1031.628,-50.727,414.434,167.895,41.884,157.787
C07831=1031.634,-50.478,414.422,167.898,41.883,157.787
C07832=1031.640,-50.229,414.409,167.901,41.882,157.787
C07833=1031.647,-49.979,414.397,167.904,41.881,157.787
C07834=1031.653,-49.730,414.384,167.907,41.880,157.787
C07835=1031.658,-49.480,414.372,167.909,41.879,157.787
C07836=1031.664,-49.230,414.359,167.911,41.877,157.786
C07837=1031.671,-48.980,414.347,167.914,41.876,157.786
C07838=1031.677,-48.730,414.335,167.917,41.875,157.786
C07839=1031.683,-48.480,414.322,167.920,41.874,157.786
C07840=1031.689,-48.232,414.311,167.923,41.873,157.786
C07841=1031.695,-47.982,414.297,167.925,41.872,157.786
C07842=1031.701,-47.732,414.285,167.928,41.871,157.786
C07843=1031.708,-47.483,414.273,167.930,41.869,157.786
C07844=1031.714,-47.233,414.260,167.933,41.868,157.786
C07845=1031.719,-46.983,414.248,167.936,41.867,157.786
C07846=1031.726,-46.733,414.236,167.938,41.866,157.786
C07847=1031.732,-46.484,414.222,167.941,41.865,157.786
C07848=1031.738,-46.234,414.210,167.944,41.864,157.786
C07849=1031.745,-45.985,414.198,167.947,41.863,157.786
C07850=1031.751,-45.735,414.185,167.949,41.861,157.786
C07851=1031.757,-45.486,414.172,167.951,41.860,157.786
C07852=1031.764,-45.236,414.160,167.954,41.859,157.786
C07853=1031.770,-44.986,414.148,167.957,41.858,157.786
C07854=1031.775,-44.736,414.135,167.960,41.857,157.786
C07855=1031.782,-44.487,414.122,167.962,41.856,157.786
C07856=1031.788,-44.237,414.110,167.964,41.855,157.786
C07857=1031.794,-43.988,414.097,167.967,41.853,157.786
C07858=1031.800,-43.738,414.085,167.970,41.852,157.786
C07859=1031.807,-43.489,414.072,167.973,41.851,157.786
C07860=1031.813,-43.239,414.059,167.975,41.850,157.786
C07861=1031.819,-42.989,414.047,167.978,41.849,157.786
C07862=1031.826,-42.740,414.034,167.980,41.848,157.785
C07863=1031.832,-42.490,414.022,167.983,41.847,157.785
C07864=1031.838,-42.240,414.009,167.986,41.845,157.785
C07865=1031.844,-41.991,413.996,167.988,41.844,157.785
C07866=1031.851,-41.741,413.984,167.991,41.843,157.785
C07867=1031.857,-41.492,413.971,167.994,41.842,157.785
C07868=1031.863,-41.242,413.958,167.997,41.841,157.785
C07869=1031.869,-40.993,413.946,167.999,41.840,157.785
C07870=1031.876,-40.743,413.933,168.001,41.838,157.785
C07871=1031.881,-40.494,413.920,168.004,41.837,157.785
C07872=1031.887,-40.244,413.908,168.007,41.836,157.785
C07873=1031.894,-39.995,413.895,168.010,41.835,157.785
C07874=1031.900,-39.745,413.883,168.012,41.834,157.785
C07875=1031.906,-39.496,413.869,168.014,41.833,157.785
C07876=1031.912,-39.246,413.857,168.017,41.831,157.785
C07877=1031.919,-38.997,413.844,168.020,41.830,157.785
C07878=1031.926,-38.746,413.831,168.023,41.829,157.785
C07879=1031.932,-38.497,413.818,168.025,41.828,157.785
C07880=1031.938,-38.247,413.805,168.028,41.827,157.785
C07881=1031.944,-37.998,413.792,168.030,41.826,157.785
C07882=1031.950,-37.748,413.779,168.032,41.825,157.785
C07883=1031.956,-37.499,413.766,168.035,41.824,157.785
C07884=1031.962,-37.249,413.754,168.038,41.823,157.785
C07885=1031.968,-36.999,413.740,168.041,41.822,157.785
C07886=1031.975,-36.750,413.727,168.043,41.821,157.784
C07887=1031.982,-36.469,413.713,168.046,41.820,157.784
C07888=1031.989,-36.188,413.699,168.049,41.819,157.784
C07889=1031.995,-35.908,413.683,168.051,41.817,157.784
C07890=1032.002,-35.626,413.669,168.055,41.816,157.784
C07891=1032.009,-35.377,413.656,168.057,41.815,157.784
C07892=1032.015,-35.128,413.642,168.060,41.814,157.784
C07893=1032.021,-34.878,413.630,168.063,41.813,157.784
C07894=1032.027,-34.629,413.616,168.065,41.812,157.784
C07895=1032.034,-34.379,413.603,168.067,41.811,157.784
C07896=1032.040,-34.129,413.590,168.070,41.809,157.784
C07897=1032.046,-33.879,413.577,168.073,41.808,157.784
C07898=1032.052,-33.630,413.564,168.075,41.807,157.784
C07899=1032.058,-33.380,413.551,168.078,41.806,157.784
C07900=1032.064,-33.131,413.538,168.081,41.805,157.784
C07901=1032.071,-32.881,413.524,168.083,41.804,157.784
C07902=1032.077,-32.631,413.512,168.086,41.803,157.784
C07903=1032.083,-32.382,413.498,168.088,41.802,157.784
C07904=1032.089,-32.133,413.485,168.091,41.801,157.784
C07905=1032.096,-31.883,413.472,168.093,41.800,157.784
C07906=1032.102,-31.633,413.459,168.096,41.799,157.784
C07907=1032.108,-31.384,413.446,168.099,41.798,157.784
C07908=1032.115,-31.134,413.432,168.101,41.797,157.784
C07909=1032.121,-30.885,413.419,168.104,41.796,157.784
C07910=1032.127,-30.634,413.406,168.107,41.795,157.784
C07911=1032.133,-30.385,413.393,168.108,41.794,157.784
C07912=1032.140,-30.136,413.380,168.111,41.793,157.784
C07913=1032.146,-29.887,413.366,168.114,41.792,157.784
C07914=1032.153,-29.637,413.353,168.117,41.791,157.784
C07915=1032.159,-29.387,413.340,168.119,41.790,157.784
C07916=1032.165,-29.138,413.327,168.122,41.788,157.783
C07917=1032.171,-28.888,413.314,168.124,41.787,157.783
C07918=1032.178,-28.638,413.300,168.126,41.786,157.783
C07919=1032.184,-28.389,413.287,168.129,41.785,157.783
C07920=1032.190,-28.140,413.274,168.132,41.784,157.783
C07921=1032.197,-27.890,413.260,168.135,41.783,157.783
C07922=1032.203,-27.640,413.247,168.137,41.782,157.783
C07923=1032.209,-27.391,413.234,168.140,41.781,157.783
C07924=1032.215,-27.141,413.221,168.142,41.780,157.783
C07925=1032.221,-26.891,413.207,168.144,41.779,157.783
C07926=1032.228,-26.642,413.193,168.147,41.778,157.783
C07927=1032.234,-26.393,413.180,168.150,41.777,157.783
C07928=1032.240,-26.142,413.166,168.152,41.776,157.783
C07929=1032.246,-25.893,413.153,168.155,41.775,157.783
C07930=1032.252,-25.644,413.139,168.157,41.775,157.783
C07931=1032.259,-25.393,413.125,168.160,41.773,157.783
C07932=1032.265,-25.144,413.112,168.163,41.772,157.783
C07933=1032.271,-24.895,413.099,168.164,41.771,157.783
C07934=1032.277,-24.646,413.085,168.167,41.770,157.783
C07935=1032.283,-24.395,413.071,168.170,41.769,157.783
C07936=1032.289,-24.146,413.058,168.172,41.768,157.783
C07937=1032.296,-23.897,413.044,168.175,41.767,157.783
C07938=1032.302,-23.647,413.030,168.178,41.766,157.783
C07939=1032.308,-23.398,413.016,168.180,41.765,157.783
C07940=1032.314,-23.149,413.003,168.183,41.765,157.783
C07941=1032.321,-22.899,412.989,168.185,41.764,157.783
C07942=1032.327,-22.649,412.975,168.187,41.763,157.783
C07943=1032.334,-22.334,412.958,168.190,41.762,157.783
C07944=1032.343,-22.019,412.941,168.194,41.760,157.783
C07945=1032.351,-21.704,412.924,168.197,41.759,157.783
C07946=1032.359,-21.389,412.907,168.200,41.758,157.783
C07947=1032.364,-21.156,412.894,168.203,41.757,157.783
C07948=1032.370,-20.923,412.881,168.204,41.756,157.783
C07949=1032.376,-20.690,412.868,168.207,41.755,157.783
C07950=1032.382,-20.458,412.855,168.209,41.754,157.783
C07951=1032.388,-20.225,412.842,168.212,41.753,157.783
C07952=1032.394,-19.992,412.829,168.214,41.752,157.783
C07953=1032.400,-19.759,412.817,168.217,41.751,157.783
C07954=1032.405,-19.526,412.804,168.219,41.750,157.783
C07955=1032.412,-19.277,412.791,168.222,41.749,157.783
C07956=1032.418,-19.027,412.776,168.224,41.748,157.782
C07957=1032.424,-18.778,412.763,168.226,41.747,157.782
C07958=1032.431,-18.528,412.749,168.228,41.746,157.782
C07959=1032.436,-18.278,412.735,168.231,41.745,157.782
C07960=1032.443,-18.029,412.721,168.234,41.744,157.782
C07961=1032.450,-17.780,412.707,168.236,41.743,157.782
C07962=1032.455,-17.530,412.694,168.239,41.742,157.782
C07963=1032.462,-17.280,412.680,168.242,41.742,157.782
C07964=1032.469,-17.031,412.666,168.244,41.741,157.782
C07965=1032.475,-16.781,412.652,168.247,41.740,157.782
C07966=1032.481,-16.532,412.638,168.248,41.739,157.782
C07967=1032.488,-16.282,412.624,168.251,41.738,157.782
C07968=1032.494,-16.033,412.610,168.254,41.737,157.782
C07969=1032.500,-15.783,412.597,168.256,41.736,157.782
C07970=1032.507,-15.534,412.583,168.259,41.735,157.782
C07971=1032.513,-15.284,412.568,168.261,41.734,157.782
C07972=1032.519,-15.035,412.555,168.264,41.733,157.782
C07973=1032.526,-14.785,412.540,168.266,41.732,157.782
C07974=1032.531,-14.535,412.526,168.269,41.732,157.782
C07975=1032.538,-14.286,412.513,168.271,41.731,157.782
C07976=1032.544,-14.037,412.498,168.273,41.730,157.782
C07977=1032.550,-13.787,412.484,168.276,41.729,157.782
C07978=1032.556,-13.538,412.470,168.278,41.728,157.782
C07979=1032.562,-13.287,412.456,168.281,41.727,157.782
C07980=1032.569,-13.038,412.441,168.284,41.726,157.782
C07981=1032.575,-12.788,412.427,168.286,41.725,157.782
C07982=1032.582,-12.539,412.413,168.289,41.724,157.782
C07983=1032.587,-12.290,412.399,168.290,41.723,157.782
C07984=1032.594,-12.040,412.384,168.293,41.722,157.782
C07985=1032.600,-11.791,412.371,168.295,41.722,157.782
C07986=1032.606,-11.541,412.356,168.298,41.721,157.782
C07987=1032.613,-11.292,412.343,168.300,41.720,157.782
C07988=1032.619,-11.042,412.328,168.303,41.719,157.782
C07989=1032.625,-10.792,412.314,168.306,41.718,157.782
C07990=1032.632,-10.543,412.300,168.308,41.717,157.782
C07991=1032.638,-10.293,412.285,168.311,41.716,157.782
C07992=1032.644,-10.044,412.271,168.313,41.715,157.782
C07993=1032.651,-9.795,412.256,168.315,41.714,157.782
C07994=1032.656,-9.545,412.243,168.317,41.713,157.782
C07995=1032.663,-9.296,412.228,168.320,41.712,157.782
C07996=1032.669,-9.045,412.214,168.322,41.711,157.782
C07997=1032.675,-8.796,412.199,168.325,41.710,157.782
C07998=1032.682,-8.546,412.186,168.327,41.710,157.782
C07999=1032.688,-8.297,412.171,168.330,41.709,157.782
C08000=1032.694,-8.048,412.156,168.333,41.708,157.782
C08001=1032.701,-7.798,412.143,168.335,41.707,157.782
C08002=1032.707,-7.549,412.128,168.337,41.706,157.782
C08003=1032.714,-7.300,412.114,168.339,41.705,157.782
C08004=1032.720,-7.049,412.099,168.342,41.704,157.782
C08005=1032.726,-6.800,412.085,168.344,41.704,157.782
C08006=1032.733,-6.551,412.071,168.347,41.703,157.782
C08007=1032.738,-6.301,412.057,168.349,41.702,157.782
C08008=1032.745,-6.052,412.042,168.352,41.701,157.782
C08009=1032.752,-5.802,412.027,168.354,41.700,157.781
C08010=1032.757,-5.553,412.014,168.357,41.699,157.781
C08011=1032.764,-5.303,411.999,168.359,41.698,157.781
C08012=1032.771,-5.054,411.984,168.361,41.697,157.781
C08013=1032.777,-4.804,411.970,168.364,41.696,157.781
C08014=1032.783,-4.555,411.956,168.366,41.695,157.781
C08015=1032.790,-4.271,411.940,168.369,41.694,157.781
C08016=1032.798,-3.989,411.923,168.372,41.693,157.781
C08017=1032.805,-3.705,411.906,168.375,41.692,157.781
C08018=1032.812,-3.422,411.890,168.378,41.691,157.781
C08019=1032.818,-3.172,411.875,168.380,41.690,157.781
C08020=1032.824,-2.923,411.860,168.383,41.690,157.781
C08021=1032.831,-2.673,411.845,168.384,41.689,157.781
C08022=1032.837,-2.424,411.830,168.387,41.688,157.781
C08023=1032.843,-2.175,411.816,168.389,41.688,157.781
C08024=1032.849,-1.925,411.801,168.391,41.687,157.781
C08025=1032.855,-1.675,411.786,168.394,41.686,157.781
C08026=1032.861,-1.426,411.772,168.396,41.685,157.781
C08027=1032.867,-1.176,411.757,168.399,41.684,157.781
C08028=1032.874,-0.927,411.742,168.401,41.683,157.781
C08029=1032.879,-0.678,411.728,168.404,41.683,157.781
C08030=1032.886,-0.428,411.713,168.406,41.682,157.781
C08031=1032.892,-0.178,411.698,168.409,41.681,157.781
C08032=1032.899,0.071,411.683,168.410,41.680,157.781
C08033=1032.904,0.320,411.668,168.413,41.680,157.781
C08034=1032.911,0.570,411.653,168.415,41.679,157.781
C08035=1032.917,0.820,411.638,168.418,41.678,157.781
C08036=1032.924,1.069,411.623,168.420,41.677,157.781
C08037=1032.929,1.318,411.609,168.423,41.676,157.781
C08038=1032.936,1.568,411.594,168.425,41.675,157.781
C08039=1032.942,1.818,411.579,168.427,41.675,157.781
C08040=1032.948,2.067,411.564,168.430,41.674,157.781
C08041=1032.954,2.316,411.549,168.432,41.673,157.781
C08042=1032.961,2.566,411.534,168.435,41.672,157.781
C08043=1032.967,2.816,411.520,168.437,41.672,157.781
C08044=1032.973,3.065,411.505,168.440,41.671,157.781
C08045=1032.979,3.314,411.490,168.441,41.670,157.781
C08046=1032.986,3.564,411.475,168.444,41.669,157.781
C08047=1032.992,3.813,411.460,168.446,41.669,157.781
C08048=1032.998,4.063,411.445,168.449,41.667,157.781
C08049=1033.005,4.313,411.430,168.451,41.667,157.781
C08050=1033.011,4.561,411.415,168.453,41.666,157.781
C08051=1033.017,4.811,411.400,168.456,41.665,157.781
C08052=1033.024,5.060,411.385,168.458,41.664,157.781
C08053=1033.030,5.310,411.370,168.461,41.663,157.781
C08054=1033.036,5.560,411.355,168.463,41.663,157.781
C08055=1033.043,5.809,411.340,168.466,41.662,157.781
C08056=1033.049,6.058,411.326,168.467,41.661,157.781
C08057=1033.055,6.308,411.311,168.470,41.660,157.781
C08058=1033.062,6.557,411.295,168.472,41.660,157.781
C08059=1033.068,6.807,411.280,168.475,41.659,157.781
C08060=1033.074,7.056,411.265,168.477,41.658,157.781
C08061=1033.081,7.306,411.250,168.480,41.657,157.781
C08062=1033.087,7.556,411.235,168.482,41.656,157.781
C08063=1033.093,7.805,411.220,168.484,41.655,157.781
C08064=1033.100,8.054,411.205,168.487,41.654,157.781
C08065=1033.106,8.303,411.190,168.488,41.653,157.781
C08066=1033.112,8.553,411.175,168.492,41.653,157.781
C08067=1033.119,8.803,411.160,168.493,41.652,157.781
C08068=1033.125,9.052,411.144,168.496,41.651,157.781
C08069=1033.132,9.301,411.130,168.498,41.650,157.781
C08070=1033.138,9.551,411.115,168.501,41.649,157.781
C08071=1033.144,9.801,411.099,168.503,41.649,157.781
C08072=1033.150,10.051,411.084,168.505,41.648,157.781
C08073=1033.157,10.300,411.068,168.508,41.647,157.781
C08074=1033.163,10.549,411.053,168.510,41.646,157.781
C08075=1033.169,10.798,411.039,168.513,41.645,157.781
C08076=1033.176,11.047,411.023,168.515,41.645,157.781
C08077=1033.182,11.297,411.008,168.517,41.644,157.781
C08078=1033.189,11.547,410.993,168.519,41.643,157.781
C08079=1033.196,11.832,410.976,168.522,41.642,157.781
C08080=1033.204,12.117,410.958,168.525,41.640,157.781
C08081=1033.210,12.402,410.941,168.528,41.639,157.781
C08082=1033.218,12.687,410.924,168.530,41.638,157.781
C08083=1033.224,12.936,410.908,168.533,41.638,157.781
C08084=1033.231,13.186,410.893,168.535,41.637,157.781
C08085=1033.237,13.436,410.878,168.537,41.636,157.781
C08086=1033.244,13.685,410.863,168.539,41.635,157.781
C08087=1033.250,13.934,410.848,168.542,41.634,157.781
C08088=1033.257,14.184,410.833,168.544,41.634,157.781
C08089=1033.263,14.433,410.816,168.546,41.633,157.781
C08090=1033.269,14.683,410.801,168.549,41.632,157.781
C08091=1033.276,14.932,410.786,168.551,41.632,157.781
C08092=1033.281,15.182,410.770,168.554,41.631,157.781
C08093=1033.288,15.431,410.755,168.556,41.630,157.781
C08094=1033.294,15.681,410.740,168.558,41.629,157.781
C08095=1033.300,15.930,410.723,168.561,41.628,157.781
C08096=1033.307,16.180,410.708,168.563,41.628,157.781
C08097=1033.313,16.429,410.693,168.566,41.627,157.781
C08098=1033.319,16.679,410.677,168.567,41.626,157.781
C08099=1033.326,16.928,410.662,168.569,41.625,157.781
C08100=1033.332,17.177,410.647,168.572,41.625,157.781
C08101=1033.338,17.427,410.630,168.574,41.624,157.781
C08102=1033.344,17.677,410.615,168.577,41.623,157.781
C08103=1033.351,17.926,410.600,168.579,41.623,157.781
C08104=1033.357,18.175,410.583,168.581,41.622,157.781
C08105=1033.364,18.425,410.569,168.584,41.621,157.781
C08106=1033.370,18.674,410.553,168.586,41.620,157.781
C08107=1033.376,18.924,410.537,168.588,41.619,157.781
C08108=1033.383,19.173,410.522,168.591,41.618,157.781
C08109=1033.389,19.422,410.507,168.593,41.618,157.781
C08110=1033.395,19.672,410.490,168.595,41.617,157.781
C08111=1033.402,19.921,410.474,168.597,41.616,157.781
C08112=1033.408,20.171,410.459,168.599,41.616,157.781
C08113=1033.414,20.420,410.443,168.602,41.615,157.781
C08114=1033.420,20.670,410.427,168.604,41.614,157.780
C08115=1033.427,20.919,410.412,168.606,41.614,157.781
C08116=1033.434,21.168,410.396,168.609,41.613,157.781
C08117=1033.439,21.418,410.380,168.611,41.612,157.781
C08118=1033.446,21.667,410.365,168.614,41.611,157.781
C08119=1033.452,21.917,410.349,168.616,41.610,157.781
C08120=1033.458,22.166,410.333,168.618,41.610,157.781
C08121=1033.464,22.415,410.317,168.621,41.609,157.781
C08122=1033.471,22.665,410.302,168.622,41.608,157.780
C08123=1033.477,22.914,410.286,168.624,41.608,157.781
C08124=1033.484,23.164,410.270,168.627,41.607,157.781
C08125=1033.490,23.413,410.253,168.629,41.606,157.780
C08126=1033.496,23.663,410.239,168.631,41.606,157.781
C08127=1033.502,23.912,410.222,168.634,41.604,157.781
C08128=1033.509,24.161,410.207,168.636,41.604,157.780
C08129=1033.515,24.411,410.190,168.639,41.603,157.781
C08130=1033.521,24.660,410.175,168.641,41.602,157.780
C08131=1033.527,24.910,410.159,168.643,41.601,157.780
C08132=1033.535,25.159,410.143,168.646,41.601,157.781
C08133=1033.541,25.409,410.127,168.648,41.600,157.780
C08134=1033.547,25.658,410.111,168.649,41.599,157.780
C08135=1033.553,25.908,410.096,168.653,41.599,157.781
C08136=1033.560,26.157,410.080,168.654,41.598,157.780
C08137=1033.566,26.406,410.064,168.656,41.597,157.780
C08138=1033.573,26.656,410.048,168.659,41.596,157.781
C08139=1033.579,26.905,410.031,168.661,41.596,157.780
C08140=1033.585,27.155,410.015,168.664,41.595,157.781
C08141=1033.591,27.404,410.000,168.666,41.594,157.780
C08142=1033.597,27.653,409.983,168.668,41.593,157.780
C08143=1033.604,27.940,409.965,168.671,41.592,157.780
C08144=1033.612,28.226,409.947,168.674,41.592,157.780
C08145=1033.619,28.512,409.928,168.676,41.591,157.780
C08146=1033.626,28.799,409.910,168.679,41.590,157.780
C08147=1033.632,29.048,409.894,168.681,41.590,157.780
C08148=1033.639,29.298,409.878,168.683,41.589,157.780
C08149=1033.646,29.548,409.862,168.685,41.588,157.781
C08150=1033.651,29.797,409.845,168.687,41.587,157.780
C08151=1033.657,30.046,409.829,168.690,41.587,157.781
C08152=1033.664,30.295,409.813,168.692,41.586,157.780
C08153=1033.670,30.545,409.797,168.694,41.585,157.780
C08154=1033.676,30.794,409.781,168.697,41.585,157.781
C08155=1033.683,31.044,409.765,168.699,41.584,157.780
C08156=1033.689,31.293,409.749,168.701,41.584,157.781
C08157=1033.696,31.542,409.732,168.703,41.583,157.780
C08158=1033.701,31.791,409.715,168.706,41.582,157.781
C08159=1033.709,32.041,409.699,168.708,41.581,157.781
C08160=1033.715,32.290,409.683,168.710,41.580,157.780
C08161=1033.721,32.540,409.667,168.713,41.580,157.781
C08162=1033.727,32.789,409.651,168.714,41.579,157.781
C08163=1033.734,33.039,409.635,168.717,41.579,157.781
C08164=1033.740,33.288,409.618,168.719,41.578,157.781
C08165=1033.746,33.537,409.602,168.721,41.577,157.780
C08166=1033.752,33.787,409.586,168.723,41.577,157.781
C08167=1033.759,34.036,409.570,168.726,41.576,157.781
C08168=1033.765,34.285,409.553,168.728,41.575,157.781
C08169=1033.771,34.535,409.537,168.730,41.574,157.781
C08170=1033.777,34.784,409.520,168.733,41.573,157.781
C08171=1033.785,35.034,409.504,168.735,41.573,157.781
C08172=1033.790,35.283,409.488,168.737,41.572,157.781
C08173=1033.796,35.532,409.472,168.740,41.571,157.780
C08174=1033.803,35.782,409.455,168.742,41.571,157.781
C08175=1033.810,36.031,409.439,168.744,41.570,157.780
C08176=1033.816,36.280,409.423,168.747,41.570,157.781
C08177=1033.822,36.530,409.406,168.748,41.569,157.781
C08178=1033.828,36.780,409.390,168.750,41.568,157.780
C08179=1033.834,37.029,409.373,168.753,41.567,157.781
C08180=1033.842,37.278,409.357,168.755,41.566,157.781
C08181=1033.848,37.527,409.340,168.757,41.565,157.780
C08182=1033.854,37.777,409.324,168.759,41.565,157.781
C08183=1033.860,38.026,409.308,168.762,41.564,157.780
C08184=1033.867,38.275,409.291,168.764,41.564,157.781
C08185=1033.873,38.525,409.274,168.766,41.563,157.780
C08186=1033.879,38.774,409.258,168.769,41.563,157.781
C08187=1033.885,39.024,409.241,168.771,41.562,157.781
C08188=1033.891,39.273,409.224,168.773,41.561,157.781
C08189=1033.897,39.522,409.208,168.775,41.561,157.781
C08190=1033.904,39.772,409.191,168.778,41.560,157.781
C08191=1033.910,40.021,409.175,168.780,41.559,157.781
C08192=1033.916,40.270,409.158,168.782,41.559,157.781
C08193=1033.923,40.520,409.141,168.784,41.558,157.781
C08194=1033.929,40.769,409.125,168.786,41.558,157.781
C08195=1033.935,41.019,409.108,168.788,41.557,157.781
C08196=1033.942,41.268,409.091,168.790,41.556,157.781
C08197=1033.948,41.517,409.075,168.793,41.555,157.781
C08198=1033.955,41.767,409.058,168.795,41.554,157.781
C08199=1033.960,42.016,409.041,168.797,41.554,157.781
C08200=1033.966,42.265,409.025,168.800,41.553,157.781
C08201=1033.973,42.515,409.008,168.802,41.553,157.781
C08202=1033.979,42.764,408.991,168.804,41.552,157.781
C08203=1033.985,43.013,408.974,168.806,41.552,157.781
C08204=1033.992,43.263,408.958,168.809,41.551,157.781
C08205=1033.998,43.512,408.940,168.811,41.550,157.781
C08206=1034.004,43.762,408.924,168.813,41.550,157.781
C08207=1034.011,44.048,408.904,168.816,41.549,157.781
C08208=1034.018,44.335,408.884,168.818,41.549,157.781
C08209=1034.025,44.621,408.866,168.821,41.548,157.781
C08210=1034.032,44.907,408.846,168.823,41.548,157.781
C08211=1034.039,45.157,408.829,168.825,41.546,157.781
C08212=1034.044,45.406,408.812,168.827,41.546,157.781
C08213=1034.050,45.655,408.795,168.829,41.545,157.781
C08214=1034.057,45.905,408.778,168.831,41.545,157.781
C08215=1034.063,46.153,408.761,168.834,41.544,157.781
C08216=1034.069,46.404,408.744,168.836,41.544,157.781
C08217=1034.075,46.652,408.727,168.838,41.543,157.781
C08218=1034.082,46.901,408.710,168.840,41.543,157.781
C08219=1034.088,47.151,408.693,168.843,41.542,157.781
C08220=1034.094,47.400,408.676,168.845,41.541,157.781
C08221=1034.100,47.650,408.659,168.847,41.541,157.781
C08222=1034.106,47.899,408.642,168.849,41.540,157.781
C08223=1034.113,48.149,408.624,168.852,41.540,157.781
C08224=1034.119,48.398,408.608,168.854,41.539,157.781
C08225=1034.125,48.647,408.591,168.856,41.539,157.781
C08226=1034.132,48.896,408.574,168.858,41.538,157.781
C08227=1034.137,49.146,408.557,168.861,41.537,157.781
C08228=1034.144,49.395,408.539,168.863,41.537,157.781
C08229=1034.150,49.644,408.523,168.865,41.536,157.781
C08230=1034.156,49.894,408.505,168.867,41.536,157.781
C08231=1034.162,50.143,408.488,168.870,41.535,157.781
C08232=1034.169,50.393,408.471,168.872,41.534,157.781
C08233=1034.175,50.641,408.454,168.873,41.534,157.781
C08234=1034.181,50.892,408.437,168.875,41.533,157.781
C08235=1034.187,51.140,408.420,168.878,41.532,157.781
C08236=1034.194,51.390,408.402,168.880,41.532,157.781
C08237=1034.200,51.639,408.385,168.882,41.531,157.781
C08238=1034.206,51.889,408.368,168.884,41.531,157.781
C08239=1034.212,52.138,408.351,168.887,41.530,157.781
C08240=1034.219,52.387,408.333,168.889,41.530,157.781
C08241=1034.225,52.636,408.316,168.891,41.529,157.781
C08242=1034.231,52.886,408.300,168.893,41.528,157.781
C08243=1034.237,53.135,408.282,168.896,41.527,157.781
C08244=1034.244,53.385,408.265,168.898,41.527,157.781
C08245=1034.250,53.633,408.248,168.900,41.526,157.781
C08246=1034.257,53.883,408.231,168.902,41.526,157.781
C08247=1034.262,54.133,408.214,168.905,41.525,157.781
C08248=1034.269,54.382,408.196,168.907,41.525,157.781
C08249=1034.276,54.631,408.179,168.909,41.524,157.781
C08250=1034.281,54.880,408.161,168.911,41.523,157.781
C08251=1034.288,55.130,408.144,168.913,41.522,157.781
C08252=1034.294,55.379,408.127,168.915,41.522,157.781
C08253=1034.301,55.628,408.109,168.917,41.521,157.781
C08254=1034.306,55.878,408.093,168.919,41.521,157.781
C08255=1034.313,56.127,408.076,168.922,41.520,157.781
C08256=1034.319,56.377,408.058,168.924,41.520,157.782
C08257=1034.326,56.626,408.041,168.926,41.519,157.781
C08258=1034.333,56.875,408.023,168.929,41.518,157.782
C08259=1034.338,57.124,408.006,168.931,41.517,157.781
C08260=1034.345,57.373,407.988,168.933,41.516,157.781
C08261=1034.352,57.623,407.971,168.935,41.516,157.781
C08262=1034.357,57.872,407.954,168.938,41.515,157.781
C08263=1034.364,58.121,407.936,168.940,41.515,157.782
C08264=1034.370,58.371,407.920,168.942,41.514,157.781
C08265=1034.376,58.620,407.902,168.944,41.514,157.782
C08266=1034.383,58.870,407.885,168.947,41.513,157.781
C08267=1034.389,59.119,407.868,168.949,41.512,157.782
C08268=1034.395,59.368,407.850,168.950,41.511,157.781
C08269=1034.402,59.618,407.832,168.952,41.511,157.781
C08270=1034.409,59.867,407.816,168.955,41.510,157.782
C08271=1034.416,60.153,407.795,168.957,41.509,157.781
C08272=1034.423,60.439,407.775,168.960,41.509,157.782
C08273=1034.430,60.725,407.755,168.963,41.508,157.782
C08274=1034.439,61.011,407.735,168.965,41.507,157.781
C08275=1034.444,61.260,407.717,168.967,41.507,157.782
C08276=1034.451,61.509,407.700,168.970,41.506,157.781
C08277=1034.457,61.759,407.682,168.972,41.505,157.781
C08278=1034.463,62.008,407.665,168.974,41.504,157.781
C08279=1034.470,62.257,407.648,168.977,41.503,157.781
C08280=1034.476,62.507,407.630,168.979,41.503,157.782
C08281=1034.483,62.756,407.612,168.980,41.502,157.781
C08282=1034.490,63.005,407.595,168.982,41.501,157.781
C08283=1034.496,63.255,407.578,168.985,41.501,157.781
C08284=1034.503,63.504,407.560,168.987,41.500,157.781
C08285=1034.508,63.753,407.543,168.989,41.500,157.781
C08286=1034.515,64.003,407.525,168.991,41.499,157.781
C08287=1034.521,64.252,407.507,168.994,41.498,157.782
C08288=1034.528,64.501,407.489,168.996,41.498,157.781
C08289=1034.534,64.750,407.472,168.998,41.497,157.782
C08290=1034.540,65.000,407.454,169.000,41.497,157.782
C08291=1034.547,65.249,407.436,169.003,41.496,157.782
C08292=1034.552,65.498,407.419,169.005,41.496,157.782
C08293=1034.559,65.748,407.400,169.007,41.495,157.782
C08294=1034.565,65.997,407.383,169.009,41.495,157.782
C08295=1034.571,66.246,407.365,169.012,41.494,157.782
C08296=1034.578,66.495,407.348,169.014,41.493,157.782
C08297=1034.584,66.745,407.329,169.016,41.492,157.782
C08298=1034.590,66.994,407.311,169.018,41.492,157.782
C08299=1034.596,67.243,407.294,169.019,41.491,157.782
C08300=1034.603,67.493,407.277,169.023,41.491,157.782
C08301=1034.609,67.742,407.258,169.025,41.491,157.782
C08302=1034.615,67.992,407.240,169.026,41.490,157.782
C08303=1034.622,68.240,407.223,169.028,41.489,157.782
C08304=1034.628,68.490,407.204,169.031,41.488,157.782
C08305=1034.634,68.739,407.186,169.033,41.488,157.782
C08306=1034.641,68.989,407.169,169.035,41.487,157.782
C08307=1034.647,69.237,407.151,169.037,41.487,157.782
C08308=1034.653,69.487,407.133,169.040,41.486,157.782
C08309=1034.659,69.737,407.115,169.042,41.486,157.782
C08310=1034.665,69.986,407.096,169.044,41.485,157.782
C08311=1034.672,70.234,407.079,169.046,41.484,157.782
C08312=1034.678,70.484,407.061,169.048,41.484,157.782
C08313=1034.684,70.733,407.043,169.051,41.483,157.782
C08314=1034.690,70.983,407.025,169.053,41.483,157.782
C08315=1034.696,71.231,407.006,169.055,41.483,157.782
C08316=1034.702,71.481,406.989,169.057,41.482,157.782
C08317=1034.710,71.730,406.970,169.060,41.481,157.782
C08318=1034.716,71.980,406.953,169.062,41.480,157.782
C08319=1034.722,72.229,406.934,169.064,41.480,157.782
C08320=1034.728,72.478,406.916,169.066,41.480,157.782
C08321=1034.734,72.728,406.898,169.068,41.479,157.782
C08322=1034.740,72.977,406.880,169.071,41.479,157.782
C08323=1034.746,73.227,406.862,169.072,41.478,157.782
C08324=1034.753,73.476,406.843,169.075,41.477,157.782
C08325=1034.759,73.724,406.826,169.077,41.477,157.782
C08326=1034.765,73.974,406.808,169.079,41.476,157.782
C08327=1034.771,74.223,406.790,169.081,41.476,157.782
C08328=1034.778,74.472,406.771,169.083,41.475,157.782
C08329=1034.784,74.722,406.753,169.085,41.475,157.782
C08330=1034.790,74.971,406.734,169.087,41.474,157.782
C08331=1034.796,75.220,406.716,169.090,41.473,157.782
C08332=1034.802,75.469,406.698,169.092,41.473,157.782
C08333=1034.810,75.718,406.680,169.094,41.472,157.782
C08334=1034.816,75.968,406.662,169.096,41.472,157.782
C08335=1034.822,76.254,406.641,169.099,41.471,157.782
C08336=1034.830,76.540,406.620,169.101,41.471,157.782
C08337=1034.837,76.825,406.599,169.104,41.470,157.782
C08338=1034.844,77.111,406.578,169.107,41.469,157.782
C08339=1034.851,77.361,406.560,169.109,41.468,157.782
C08340=1034.856,77.609,406.541,169.111,41.468,157.782
C08341=1034.863,77.859,406.523,169.113,41.468,157.782
C08342=1034.869,78.108,406.505,169.115,41.467,157.782
C08343=1034.875,78.357,406.486,169.118,41.466,157.783
C08344=1034.882,78.607,406.468,169.120,41.466,157.783
C08345=1034.888,78.856,406.450,169.122,41.465,157.783
C08346=1034.894,79.105,406.431,169.124,41.465,157.783
C08347=1034.900,79.355,406.412,169.126,41.465,157.783
C08348=1034.906,79.604,406.394,169.129,41.464,157.783
C08349=1034.912,79.853,406.375,169.131,41.464,157.783
C08350=1034.918,80.102,406.357,169.133,41.463,157.783
C08351=1034.925,80.351,406.338,169.134,41.462,157.783
C08352=1034.931,80.601,406.320,169.136,41.462,157.783
C08353=1034.937,80.850,406.302,169.139,41.462,157.783
C08354=1034.943,81.099,406.282,169.142,41.461,157.783
C08355=1034.950,81.349,406.264,169.143,41.461,157.783
C08356=1034.956,81.598,406.246,169.145,41.460,157.783
C08357=1034.961,81.847,406.227,169.148,41.460,157.783
C08358=1034.968,82.096,406.209,169.150,41.459,157.783
C08359=1034.974,82.345,406.190,169.152,41.459,157.783
C08360=1034.980,82.594,406.171,169.154,41.458,157.783
C08361=1034.986,82.844,406.152,169.156,41.458,157.783
C08362=1034.993,83.093,406.134,169.159,41.457,157.783
C08363=1034.999,83.342,406.116,169.161,41.456,157.783
C08364=1035.005,83.592,406.097,169.163,41.456,157.783
C08365=1035.012,83.841,406.078,169.165,41.456,157.783
C08366=1035.018,84.090,406.060,169.167,41.455,157.783
C08367=1035.024,84.339,406.041,169.170,41.454,157.783
C08368=1035.030,84.588,406.022,169.172,41.454,157.783
C08369=1035.036,84.838,406.004,169.174,41.453,157.783
C08370=1035.043,85.087,405.985,169.176,41.453,157.783
C08371=1035.049,85.336,405.967,169.179,41.453,157.783
C08372=1035.055,85.586,405.947,169.181,41.452,157.783
C08373=1035.061,85.835,405.929,169.183,41.451,157.783
C08374=1035.068,86.084,405.910,169.185,41.451,157.783
C08375=1035.074,86.333,405.891,169.188,41.450,157.783
C08376=1035.081,86.582,405.873,169.190,41.450,157.783
C08377=1035.087,86.831,405.854,169.192,41.449,157.783
C08378=1035.093,87.081,405.835,169.194,41.449,157.783
C08379=1035.099,87.330,405.816,169.196,41.448,157.784
C08380=1035.106,87.579,405.798,169.199,41.447,157.783
C08381=1035.112,87.828,405.779,169.201,41.447,157.784
C08382=1035.119,88.077,405.760,169.202,41.446,157.783
C08383=1035.124,88.327,405.741,169.204,41.446,157.784
C08384=1035.130,88.576,405.723,169.208,41.446,157.784
C08385=1035.137,88.826,405.704,169.209,41.445,157.784
C08386=1035.143,89.075,405.686,169.211,41.444,157.784
C08387=1035.150,89.323,405.666,169.213,41.444,157.784
C08388=1035.156,89.573,405.647,169.216,41.443,157.784
C08389=1035.162,89.822,405.629,169.218,41.443,157.784
C08390=1035.168,90.071,405.610,169.220,41.442,157.784
C08391=1035.174,90.320,405.591,169.222,41.442,157.784
C08392=1035.181,90.569,405.572,169.225,41.441,157.784
C08393=1035.187,90.819,405.553,169.227,41.440,157.784
C08394=1035.193,91.068,405.534,169.229,41.440,157.784
C08395=1035.199,91.317,405.515,169.231,41.440,157.784
C08396=1035.205,91.567,405.496,169.233,41.440,157.784
C08397=1035.212,91.815,405.477,169.236,41.439,157.784
C08398=1035.217,92.064,405.458,169.238,41.438,157.784
C08399=1035.224,92.351,405.436,169.240,41.438,157.784
C08400=1035.232,92.637,405.414,169.243,41.438,157.784
C08401=1035.238,92.922,405.392,169.245,41.437,157.784
C08402=1035.246,93.208,405.370,169.248,41.436,157.784
C08403=1035.252,93.457,405.351,169.250,41.436,157.784
C08404=1035.258,93.706,405.332,169.252,41.435,157.784
C08405=1035.264,93.956,405.314,169.255,41.435,157.784
C08406=1035.270,94.204,405.294,169.257,41.435,157.784
C08407=1035.277,94.453,405.275,169.259,41.434,157.784
C08408=1035.282,94.703,405.256,169.261,41.433,157.784
C08409=1035.289,94.953,405.237,169.263,41.433,157.784
C08410=1035.295,95.202,405.217,169.266,41.433,157.784
C08411=1035.302,95.451,405.198,169.268,41.432,157.784
C08412=1035.308,95.700,405.179,169.270,41.432,157.784
C08413=1035.314,95.949,405.160,169.272,41.431,157.785
C08414=1035.320,96.198,405.140,169.275,41.430,157.785
C08415=1035.326,96.447,405.122,169.277,41.430,157.785
C08416=1035.332,96.697,405.102,169.279,41.430,157.785
C08417=1035.339,96.946,405.083,169.281,41.430,157.785
C08418=1035.345,97.195,405.063,169.284,41.429,157.785
C08419=1035.352,97.444,405.045,169.286,41.428,157.785
C08420=1035.358,97.693,405.025,169.288,41.428,157.785
C08421=1035.364,97.942,405.006,169.290,41.427,157.785
C08422=1035.370,98.192,404.987,169.293,41.427,157.785
C08423=1035.376,98.440,404.967,169.295,41.427,157.785
C08424=1035.383,98.690,404.948,169.296,41.426,157.785
C08425=1035.389,98.939,404.929,169.298,41.425,157.785
C08426=1035.395,99.188,404.909,169.302,41.425,157.785
C08427=1035.402,99.437,404.891,169.303,41.424,157.785
C08428=1035.407,99.687,404.871,169.305,41.424,157.785
C08429=1035.414,99.935,404.852,169.307,41.424,157.785
C08430=1035.420,100.185,404.832,169.310,41.422,157.785
C08431=1035.426,100.434,404.812,169.312,41.422,157.785
C08432=1035.433,100.683,404.794,169.314,41.422,157.785
C08433=1035.439,100.932,404.774,169.316,41.422,157.785
C08434=1035.444,101.182,404.755,169.318,41.421,157.785
C08435=1035.450,101.430,404.735,169.321,41.421,157.785
C08436=1035.457,101.680,404.716,169.323,41.420,157.785
C08437=1035.463,101.929,404.696,169.325,41.420,157.785
C08438=1035.469,102.179,404.676,169.327,41.420,157.785
C08439=1035.475,102.427,404.656,169.330,41.419,157.786
C08440=1035.481,102.677,404.637,169.332,41.419,157.786
C08441=1035.488,102.926,404.617,169.334,41.418,157.786
C08442=1035.494,103.175,404.598,169.336,41.418,157.786
C08443=1035.500,103.424,404.578,169.338,41.418,157.786
C08444=1035.506,103.673,404.558,169.341,41.417,157.786
C08445=1035.512,103.922,404.540,169.343,41.417,157.786
C08446=1035.519,104.172,404.519,169.345,41.416,157.786
C08447=1035.524,104.421,404.500,169.347,41.416,157.786
C08448=1035.530,104.670,404.480,169.350,41.415,157.786
C08449=1035.536,104.919,404.461,169.352,41.415,157.786
C08450=1035.543,105.168,404.442,169.354,41.414,157.786
C08451=1035.549,105.417,404.421,169.356,41.414,157.786
C08452=1035.555,105.667,404.402,169.359,41.414,157.786
C08453=1035.561,105.916,404.382,169.361,41.413,157.786
C08454=1035.567,106.164,404.362,169.363,41.413,157.786
C08455=1035.574,106.414,404.343,169.365,41.412,157.786
C08456=1035.580,106.663,404.323,169.368,41.412,157.786
C08457=1035.586,106.912,404.303,169.370,41.412,157.786
C08458=1035.592,107.161,404.284,169.372,41.411,157.786
C08459=1035.599,107.410,404.264,169.374,41.410,157.786
C08460=1035.605,107.659,404.244,169.377,41.410,157.786
C08461=1035.611,107.909,404.225,169.379,41.410,157.786
C08462=1035.617,108.158,404.205,169.381,41.409,157.786
C08463=1035.625,108.444,404.182,169.384,41.408,157.786
C08464=1035.632,108.730,404.159,169.386,41.408,157.787
C08465=1035.639,109.016,404.137,169.389,41.408,157.787
C08466=1035.646,109.302,404.114,169.392,41.407,157.787
C08467=1035.652,109.550,404.095,169.394,41.407,157.787
C08468=1035.658,109.799,404.075,169.396,41.406,157.787
C08469=1035.665,110.049,404.054,169.398,41.406,157.787
C08470=1035.671,110.298,404.035,169.401,41.406,157.787
C08471=1035.677,110.547,404.015,169.403,41.405,157.787
C08472=1035.683,110.796,403.995,169.405,41.404,157.787
C08473=1035.689,111.045,403.975,169.407,41.404,157.787
C08474=1035.695,111.294,403.955,169.410,41.404,157.787
C08475=1035.702,111.544,403.935,169.412,41.404,157.787
C08476=1035.708,111.793,403.915,169.414,41.403,157.787
C08477=1035.714,112.042,403.895,169.416,41.402,157.787
C08478=1035.720,112.291,403.875,169.419,41.402,157.787
C08479=1035.726,112.540,403.855,169.421,41.402,157.787
C08480=1035.732,112.789,403.835,169.423,41.401,157.787
C08481=1035.739,113.038,403.815,169.426,41.401,157.787
C08482=1035.745,113.287,403.795,169.428,41.400,157.787
C08483=1035.751,113.536,403.775,169.430,41.400,157.787
C08484=1035.757,113.785,403.755,169.432,41.400,157.787
C08485=1035.763,114.034,403.735,169.434,41.399,157.788
C08486=1035.769,114.283,403.715,169.437,41.399,157.788
C08487=1035.775,114.533,403.694,169.439,41.399,157.788
C08488=1035.781,114.782,403.674,169.441,41.399,157.788
C08489=1035.787,115.031,403.654,169.443,41.398,157.788
C08490=1035.794,115.280,403.634,169.446,41.398,157.788
C08491=1035.799,115.529,403.613,169.448,41.398,157.788
C08492=1035.805,115.778,403.593,169.450,41.397,157.788
C08493=1035.812,116.028,403.573,169.452,41.397,157.788
C08494=1035.818,116.276,403.553,169.455,41.397,157.788
C08495=1035.823,116.525,403.532,169.457,41.396,157.788
C08496=1035.829,116.775,403.512,169.459,41.396,157.788
C08497=1035.835,117.024,403.492,169.461,41.396,157.788
C08498=1035.841,117.273,403.472,169.464,41.396,157.788
C08499=1035.847,117.522,403.451,169.466,41.395,157.789
C08500=1035.853,117.771,403.431,169.468,41.395,157.789
C08501=1035.860,118.021,403.411,169.470,41.394,157.789
C08502=1035.866,118.269,403.390,169.473,41.394,157.789
C08503=1035.871,118.518,403.369,169.475,41.394,157.789
C08504=1035.878,118.768,403.349,169.477,41.393,157.789
C08505=1035.884,119.016,403.329,169.479,41.393,157.789
C08506=1035.890,119.266,403.308,169.482,41.393,157.789
C08507=1035.896,119.515,403.288,169.484,41.392,157.789
C08508=1035.902,119.764,403.268,169.486,41.392,157.789
C08509=1035.909,120.013,403.247,169.490,41.392,157.789
C08510=1035.914,120.262,403.227,169.492,41.391,157.789
C08511=1035.921,120.511,403.206,169.494,41.391,157.789
C08512=1035.927,120.760,403.186,169.496,41.391,157.789
C08513=1035.933,121.010,403.166,169.499,41.391,157.789
C08514=1035.939,121.258,403.145,169.500,41.390,157.789
C08515=1035.945,121.507,403.125,169.503,41.389,157.789
C08516=1035.951,121.757,403.105,169.506,41.389,157.789
C08517=1035.957,122.006,403.084,169.508,41.389,157.790
C08518=1035.963,122.255,403.064,169.510,41.389,157.790
C08519=1035.970,122.503,403.043,169.512,41.388,157.790
C08520=1035.976,122.753,403.023,169.515,41.388,157.790
C08521=1035.981,123.002,403.002,169.517,41.388,157.790
C08522=1035.988,123.251,402.981,169.519,41.387,157.790
C08523=1035.994,123.500,402.961,169.522,41.387,157.790
C08524=1036.000,123.750,402.940,169.524,41.387,157.790
C08525=1036.006,123.998,402.920,169.526,41.386,157.790
C08526=1036.013,124.247,402.899,169.529,41.385,157.790
C08527=1036.020,124.533,402.876,169.531,41.385,157.790
C08528=1036.027,124.819,402.853,169.534,41.385,157.790
C08529=1036.034,125.104,402.829,169.537,41.384,157.790
C08530=1036.041,125.390,402.805,169.539,41.384,157.790
C08531=1036.047,125.639,402.785,169.542,41.384,157.790
C08532=1036.053,125.888,402.763,169.544,41.383,157.791
C08533=1036.059,126.137,402.743,169.546,41.383,157.791
C08534=1036.066,126.386,402.723,169.548,41.382,157.791
C08535=1036.072,126.635,402.702,169.551,41.382,157.791
C08536=1036.078,126.885,402.682,169.553,41.382,157.791
C08537=1036.085,127.133,402.660,169.555,41.381,157.791
C08538=1036.091,127.382,402.641,169.558,41.381,157.791
C08539=1036.097,127.632,402.620,169.560,41.381,157.791
C08540=1036.103,127.880,402.599,169.563,41.380,157.791
C08541=1036.110,128.130,402.579,169.565,41.380,157.791
C08542=1036.115,128.378,402.557,169.567,41.380,157.791
C08543=1036.122,128.628,402.537,169.570,41.379,157.791
C08544=1036.129,128.877,402.517,169.572,41.379,157.791
C08545=1036.134,129.126,402.495,169.574,41.378,157.791
C08546=1036.141,129.375,402.475,169.577,41.378,157.791
C08547=1036.148,129.624,402.454,169.579,41.378,157.791
C08548=1036.153,129.873,402.433,169.581,41.377,157.791
C08549=1036.160,130.122,402.412,169.584,41.377,157.792
C08550=1036.166,130.371,402.392,169.586,41.377,157.792
C08551=1036.173,130.620,402.371,169.588,41.376,157.792
C08552=1036.179,130.870,402.351,169.591,41.376,157.792
C08553=1036.185,131.118,402.330,169.593,41.375,157.792
C08554=1036.191,131.368,402.309,169.595,41.375,157.792
C08555=1036.197,131.617,402.287,169.598,41.375,157.792
C08556=1036.203,131.865,402.267,169.600,41.375,157.792
C08557=1036.209,132.115,402.246,169.602,41.375,157.792
C08558=1036.215,132.363,402.224,169.605,41.374,157.792
C08559=1036.222,132.612,402.203,169.607,41.374,157.792
C08560=1036.227,132.862,402.182,169.609,41.374,157.792
C08561=1036.233,133.111,402.161,169.612,41.373,157.792
C08562=1036.240,133.360,402.140,169.614,41.373,157.792
C08563=1036.245,133.609,402.120,169.616,41.373,157.793
C08564=1036.252,133.858,402.099,169.619,41.373,157.793
C08565=1036.258,134.107,402.077,169.621,41.372,157.793
C08566=1036.263,134.356,402.056,169.623,41.372,157.793
C08567=1036.270,134.605,402.035,169.626,41.372,157.793
C08568=1036.276,134.854,402.014,169.629,41.371,157.793
C08569=1036.282,135.103,401.993,169.631,41.371,157.793
C08570=1036.289,135.352,401.972,169.634,41.371,157.793
C08571=1036.295,135.601,401.950,169.636,41.371,157.793
C08572=1036.300,135.850,401.929,169.639,41.370,157.793
C08573=1036.307,136.099,401.909,169.641,41.370,157.793
C08574=1036.313,136.349,401.887,169.643,41.370,157.793
C08575=1036.319,136.597,401.866,169.646,41.369,157.793
C08576=1036.326,136.846,401.845,169.648,41.369,157.794
C08577=1036.332,137.095,401.823,169.650,41.369,157.794
C08578=1036.338,137.345,401.802,169.653,41.368,157.794
C08579=1036.344,137.593,401.782,169.655,41.368,157.794
C08580=1036.350,137.842,401.760,169.657,41.368,157.794
C08581=1036.356,138.092,401.738,169.660,41.368,157.794
C08582=1036.362,138.340,401.717,169.662,41.368,157.794
C08583=1036.369,138.589,401.696,169.665,41.367,157.794
C08584=1036.375,138.839,401.675,169.667,41.367,157.794
C08585=1036.381,139.088,401.654,169.669,41.367,157.794
C08586=1036.386,139.336,401.632,169.672,41.367,157.794
C08587=1036.392,139.586,401.611,169.674,41.366,157.794
C08588=1036.399,139.835,401.590,169.676,41.366,157.795
C08589=1036.405,140.083,401.568,169.679,41.366,157.795
C08590=1036.411,140.332,401.547,169.681,41.365,157.795
C08591=1036.418,140.617,401.522,169.685,41.366,157.795
C08592=1036.425,140.903,401.498,169.688,41.365,157.795
C08593=1036.432,141.189,401.473,169.690,41.365,157.795
C08594=1036.438,141.474,401.448,169.693,41.365,157.795
C08595=1036.445,141.723,401.426,169.695,41.364,157.795
C08596=1036.451,141.972,401.405,169.698,41.364,157.795
C08597=1036.458,142.221,401.383,169.700,41.364,157.796
C08598=1036.464,142.470,401.362,169.703,41.364,157.796
C08599=1036.469,142.719,401.341,169.705,41.364,157.796
C08600=1036.476,142.968,401.319,169.707,41.363,157.796
C08601=1036.482,143.217,401.297,169.710,41.363,157.796
C08602=1036.488,143.466,401.276,169.712,41.363,157.796
C08603=1036.493,143.715,401.254,169.715,41.362,157.796
C08604=1036.500,143.964,401.233,169.717,41.363,157.796
C08605=1036.506,144.213,401.211,169.719,41.363,157.796
C08606=1036.512,144.462,401.190,169.722,41.362,157.796
C08607=1036.518,144.712,401.168,169.724,41.362,157.796
C08608=1036.524,144.960,401.147,169.727,41.362,157.796
C08609=1036.531,145.209,401.126,169.729,41.361,157.797
C08610=1036.537,145.458,401.104,169.731,41.361,157.797
C08611=1036.543,145.707,401.082,169.734,41.361,157.797
C08612=1036.549,145.956,401.060,169.737,41.361,157.797
C08613=1036.555,146.205,401.038,169.740,41.361,157.797
C08614=1036.562,146.454,401.017,169.742,41.360,157.797
C08615=1036.567,146.703,400.995,169.745,41.360,157.797
C08616=1036.573,146.952,400.974,169.747,41.360,157.797
C08617=1036.580,147.201,400.951,169.749,41.359,157.797
C08618=1036.586,147.450,400.930,169.752,41.360,157.798
C08619=1036.592,147.699,400.908,169.754,41.359,157.798
C08620=1036.598,147.948,400.887,169.757,41.359,157.798
C08621=1036.604,148.196,400.865,169.759,41.359,157.798
C08622=1036.610,148.446,400.842,169.761,41.359,157.798
C08623=1036.616,148.695,400.821,169.764,41.359,157.798
C08624=1036.622,148.944,400.799,169.766,41.359,157.798
C08625=1036.628,149.193,400.777,169.769,41.358,157.798
C08626=1036.635,149.442,400.755,169.771,41.358,157.798
C08627=1036.641,149.691,400.733,169.775,41.358,157.798
C08628=1036.647,149.940,400.711,169.777,41.358,157.799
C08629=1036.652,150.189,400.689,169.779,41.358,157.799
C08630=1036.658,150.438,400.668,169.782,41.357,157.799
C08631=1036.665,150.686,400.645,169.784,41.358,157.799
C08632=1036.671,150.936,400.624,169.787,41.357,157.799
C08633=1036.677,151.185,400.602,169.789,41.357,157.799
C08634=1036.683,151.433,400.580,169.792,41.357,157.799
C08635=1036.689,151.683,400.557,169.794,41.357,157.799
C08636=1036.695,151.931,400.535,169.796,41.357,157.799
C08637=1036.702,152.181,400.513,169.799,41.356,157.799
C08638=1036.708,152.430,400.492,169.801,41.357,157.800
C08639=1036.714,152.678,400.470,169.804,41.356,157.800
C08640=1036.719,152.927,400.448,169.806,41.356,157.800
C08641=1036.725,153.176,400.425,169.810,41.356,157.800
C08642=1036.732,153.425,400.404,169.812,41.356,157.800
C08643=1036.738,153.674,400.381,169.815,41.356,157.800
C08644=1036.744,153.923,400.360,169.817,41.355,157.800
C08645=1036.750,154.172,400.337,169.820,41.355,157.800
C08646=1036.756,154.421,400.315,169.822,41.355,157.801
C08647=1036.763,154.669,400.293,169.825,41.355,157.801
C08648=1036.768,154.919,400.270,169.827,41.355,157.801
C08649=1036.775,155.168,400.248,169.829,41.355,157.801
C08650=1036.781,155.417,400.226,169.832,41.355,157.801
C08651=1036.786,155.666,400.203,169.834,41.355,157.801
C08652=1036.793,155.914,400.181,169.838,41.355,157.801
C08653=1036.799,156.163,400.159,169.840,41.355,157.801
C08654=1036.805,156.412,400.137,169.843,41.354,157.801
C08655=1036.811,156.697,400.112,169.846,41.354,157.802
C08656=1036.819,156.983,400.085,169.848,41.354,157.802
C08657=1036.825,157.268,400.061,169.851,41.354,157.802
C08658=1036.833,157.553,400.034,169.854,41.354,157.802
C08659=1036.839,157.802,400.013,169.857,41.354,157.802
C08660=1036.846,158.051,399.991,169.859,41.354,157.802
C08661=1036.851,158.300,399.968,169.862,41.354,157.802
C08662=1036.857,158.549,399.946,169.864,41.353,157.803
C08663=1036.864,158.797,399.924,169.868,41.354,157.803
C08664=1036.870,159.046,399.901,169.870,41.353,157.803
C08665=1036.876,159.295,399.879,169.873,41.353,157.803
C08666=1036.881,159.544,399.856,169.875,41.353,157.803
C08667=1036.888,159.793,399.834,169.878,41.353,157.803
C08668=1036.894,160.042,399.811,169.880,41.353,157.803
C08669=1036.900,160.291,399.789,169.883,41.353,157.803
C08670=1036.906,160.540,399.766,169.885,41.353,157.804
C08671=1036.911,160.789,399.743,169.887,41.353,157.804
C08672=1036.918,161.037,399.721,169.890,41.353,157.804
C08673=1036.924,161.286,399.698,169.893,41.353,157.804
C08674=1036.929,161.535,399.675,169.896,41.353,157.804
C08675=1036.935,161.784,399.652,169.898,41.353,157.804
C08676=1036.941,162.033,399.629,169.901,41.353,157.805
C08677=1036.947,162.282,399.607,169.903,41.354,157.805
C08678=1036.953,162.531,399.585,169.906,41.353,157.805
C08679=1036.958,162.780,399.562,169.908,41.354,157.805
C08680=1036.964,163.029,399.539,169.911,41.353,157.805
C08681=1036.971,163.277,399.516,169.914,41.354,157.805
C08682=1036.976,163.526,399.493,169.917,41.353,157.805
C08683=1036.982,163.775,399.470,169.919,41.354,157.806
C08684=1036.988,164.025,399.447,169.922,41.354,157.806
C08685=1036.995,164.273,399.425,169.924,41.354,157.806
C08686=1037.001,164.522,399.402,169.927,41.354,157.806
C08687=1037.006,164.771,399.379,169.929,41.354,157.806
C08688=1037.012,165.020,399.356,169.932,41.354,157.806
C08689=1037.018,165.269,399.333,169.935,41.354,157.807
C08690=1037.024,165.518,399.311,169.938,41.354,157.807
C08691=1037.030,165.767,399.288,169.940,41.354,157.807
C08692=1037.036,166.015,399.265,169.943,41.354,157.807
C08693=1037.041,166.264,399.242,169.945,41.354,157.807
C08694=1037.047,166.513,399.219,169.948,41.354,157.807
C08695=1037.054,166.763,399.196,169.950,41.354,157.807
C08696=1037.060,167.011,399.172,169.954,41.355,157.808
C08697=1037.066,167.260,399.149,169.956,41.354,157.808
C08698=1037.072,167.509,399.127,169.959,41.355,157.808
C08699=1037.077,167.757,399.104,169.961,41.354,157.808
C08700=1037.084,168.006,399.081,169.964,41.355,157.808
C08701=1037.090,168.255,399.058,169.967,41.355,157.809
C08702=1037.096,168.505,399.035,169.969,41.355,157.809
C08703=1037.102,168.753,399.012,169.972,41.355,157.809
C08704=1037.108,169.002,398.988,169.974,41.355,157.809
C08705=1037.114,169.250,398.966,169.978,41.355,157.809
C08706=1037.120,169.499,398.943,169.980,41.355,157.809
C08707=1037.126,169.749,398.920,169.983,41.355,157.809
C08708=1037.132,169.998,398.897,169.985,41.355,157.810
C08709=1037.138,170.246,398.873,169.988,41.355,157.810
C08710=1037.144,170.495,398.850,169.991,41.355,157.810
C08711=1037.150,170.743,398.828,169.994,41.355,157.810
C08712=1037.157,170.993,398.805,169.997,41.355,157.810
C08713=1037.162,171.242,398.782,169.999,41.355,157.810
C08714=1037.168,171.490,398.758,170.002,41.355,157.810
C08715=1037.174,171.739,398.735,170.004,41.355,157.811
C08716=1037.180,171.989,398.712,170.007,41.356,157.811
C08717=1037.187,172.237,398.689,170.010,41.355,157.811
C08718=1037.193,172.486,398.666,170.012,41.356,157.811
C08719=1037.200,172.771,398.639,170.016,41.356,157.811
C08720=1037.207,173.055,398.613,170.019,41.356,157.812
C08721=1037.214,173.340,398.586,170.022,41.356,157.812
C08722=1037.221,173.624,398.560,170.025,41.356,157.812
C08723=1037.226,173.873,398.537,170.028,41.356,157.812
C08724=1037.233,174.122,398.513,170.030,41.356,157.812
C08725=1037.239,174.371,398.490,170.034,41.356,157.812
C08726=1037.245,174.620,398.467,170.037,41.356,157.813
C08727=1037.252,174.869,398.443,170.039,41.356,157.813
C08728=1037.258,175.117,398.420,170.042,41.356,157.813
C08729=1037.263,175.366,398.397,170.045,41.356,157.813
C08730=1037.270,175.615,398.373,170.047,41.357,157.813
C08731=1037.276,175.864,398.350,170.050,41.356,157.813
C08732=1037.282,176.112,398.327,170.053,41.356,157.814
C08733=1037.289,176.362,398.304,170.056,41.357,157.814
C08734=1037.295,176.610,398.280,170.059,41.356,157.814
C08735=1037.301,176.859,398.257,170.061,41.357,157.814
C08736=1037.307,177.109,398.234,170.064,41.357,157.814
C08737=1037.313,177.357,398.210,170.067,41.357,157.814
C08738=1037.319,177.606,398.187,170.069,41.357,157.815
C08739=1037.325,177.855,398.163,170.072,41.357,157.815
C08740=1037.331,178.104,398.141,170.076,41.357,157.815
C08741=1037.339,178.352,398.117,170.078,41.357,157.815
C08742=1037.344,178.601,398.094,170.081,41.357,157.815
C08743=1037.351,178.850,398.070,170.084,41.357,157.815
C08744=1037.357,179.098,398.046,170.087,41.357,157.816
C08745=1037.363,179.347,398.024,170.089,41.357,157.816
C08746=1037.369,179.596,397.999,170.092,41.357,157.816
C08747=1037.375,179.845,397.977,170.096,41.358,157.816
C08748=1037.382,180.094,397.953,170.098,41.357,157.816
C08749=1037.388,180.343,397.930,170.101,41.358,157.816
C08750=1037.395,180.592,397.906,170.104,41.358,157.817
C08751=1037.401,180.840,397.882,170.106,41.358,157.817
C08752=1037.407,181.090,397.859,170.109,41.358,157.817
C08753=1037.413,181.338,397.836,170.112,41.358,157.817
C08754=1037.419,181.587,397.812,170.116,41.358,157.817
C08755=1037.426,181.836,397.789,170.118,41.358,157.818
C08756=1037.432,182.085,397.765,170.121,41.358,157.818
C08757=1037.438,182.334,397.742,170.124,41.359,157.818
C08758=1037.445,182.583,397.718,170.126,41.358,157.818
C08759=1037.451,182.831,397.694,170.129,41.359,157.818
C08760=1037.458,183.080,397.670,170.133,41.359,157.819
C08761=1037.464,183.328,397.647,170.136,41.358,157.819
C08762=1037.470,183.578,397.623,170.138,41.359,157.819
C08763=1037.476,183.826,397.599,170.141,41.359,157.819
C08764=1037.481,184.075,397.575,170.144,41.359,157.819
C08765=1037.488,184.324,397.551,170.146,41.360,157.819
C08766=1037.494,184.572,397.527,170.150,41.360,157.820
C08767=1037.500,184.821,397.503,170.153,41.360,157.820
C08768=1037.505,185.070,397.480,170.155,41.360,157.820
C08769=1037.511,185.319,397.455,170.158,41.361,157.820
C08770=1037.517,185.568,397.431,170.161,41.361,157.821
C08771=1037.523,185.817,397.407,170.164,41.361,157.821
C08772=1037.529,186.065,397.383,170.167,41.362,157.821
C08773=1037.534,186.314,397.359,170.170,41.362,157.821
C08774=1037.541,186.563,397.335,170.172,41.362,157.821
C08775=1037.546,186.811,397.311,170.175,41.362,157.822
C08776=1037.553,187.060,397.287,170.179,41.363,157.822
C08777=1037.558,187.309,397.262,170.182,41.363,157.822
C08778=1037.565,187.558,397.238,170.184,41.364,157.822
C08779=1037.570,187.806,397.214,170.187,41.364,157.823
C08780=1037.577,188.055,397.189,170.191,41.364,157.823
C08781=1037.582,188.303,397.165,170.193,41.365,157.823
C08782=1037.589,188.552,397.141,170.196,41.365,157.823
C08783=1037.596,188.837,397.114,170.199,41.365,157.824
C08784=1037.603,189.121,397.086,170.202,41.366,157.824
C08785=1037.610,189.406,397.059,170.207,41.366,157.824
C08786=1037.617,189.689,397.031,170.210,41.367,157.824
C08787=1037.623,189.938,397.006,170.212,41.367,157.825
C08788=1037.629,190.187,396.983,170.215,41.367,157.825
C08789=1037.635,190.436,396.958,170.219,41.367,157.825
C08790=1037.641,190.684,396.933,170.222,41.368,157.825
C08791=1037.647,190.933,396.909,170.224,41.368,157.825
C08792=1037.653,191.182,396.885,170.227,41.368,157.826
C08793=1037.659,191.430,396.861,170.230,41.369,157.826
C08794=1037.665,191.679,396.837,170.234,41.369,157.826
C08795=1037.672,191.928,396.811,170.236,41.369,157.826
C08796=1037.678,192.176,396.788,170.239,41.369,157.827
C08797=1037.684,192.426,396.763,170.242,41.370,157.827
C08798=1037.689,192.675,396.738,170.245,41.370,157.827
C08799=1037.696,192.923,396.714,170.249,41.371,157.827
C08800=1037.702,193.172,396.689,170.251,41.371,157.828
C08801=1037.708,193.421,396.665,170.254,41.371,157.828
C08802=1037.714,193.669,396.641,170.257,41.372,157.828
C08803=1037.721,193.918,396.616,170.261,41.372,157.828
C08804=1037.726,194.167,396.592,170.264,41.372,157.829
C08805=1037.732,194.415,396.568,170.266,41.372,157.829
C08806=1037.739,194.664,396.543,170.269,41.373,157.829
C08807=1037.745,194.913,396.519,170.272,41.373,157.829
C08808=1037.751,195.162,396.494,170.276,41.374,157.830
C08809=1037.758,195.410,396.470,170.279,41.374,157.830
C08810=1037.763,195.659,396.445,170.281,41.374,157.830
C08811=1037.770,195.908,396.421,170.284,41.375,157.830
C08812=1037.776,196.156,396.396,170.288,41.375,157.830
C08813=1037.782,196.405,396.372,170.291,41.375,157.831
C08814=1037.789,196.654,396.347,170.294,41.375,157.831
C08815=1037.794,196.903,396.322,170.297,41.376,157.831
C08816=1037.801,197.151,396.298,170.300,41.377,157.831
C08817=1037.807,197.400,396.273,170.303,41.377,157.832
C08818=1037.813,197.649,396.249,170.306,41.377,157.832
C08819=1037.820,197.898,396.224,170.309,41.377,157.832
C08820=1037.826,198.146,396.200,170.312,41.378,157.832
C08821=1037.832,198.395,396.175,170.316,41.378,157.833
C08822=1037.838,198.644,396.151,170.319,41.379,157.833
C08823=1037.845,198.931,396.121,170.322,41.379,157.833
C08824=1037.853,199.217,396.093,170.326,41.380,157.834
C08825=1037.860,199.504,396.065,170.330,41.380,157.834
C08826=1037.867,199.790,396.036,170.333,41.380,157.834
C08827=1037.874,200.039,396.012,170.336,41.381,157.834
C08828=1037.880,200.288,395.987,170.340,41.381,157.835
C08829=1037.886,200.537,395.962,170.343,41.382,157.835
C08830=1037.893,200.786,395.938,170.345,41.382,157.835
C08831=1037.899,201.034,395.912,170.348,41.382,157.835
C08832=1037.905,201.283,395.887,170.352,41.383,157.836
C08833=1037.910,201.532,395.863,170.355,41.383,157.836
C08834=1037.916,201.780,395.837,170.358,41.384,157.836
C08835=1037.923,202.029,395.812,170.361,41.384,157.836
C08836=1037.930,202.277,395.787,170.365,41.385,157.837
C08837=1037.935,202.527,395.763,170.368,41.385,157.837
C08838=1037.942,202.775,395.737,170.370,41.386,157.837
C08839=1037.947,203.023,395.712,170.374,41.387,157.838
C08840=1037.953,203.272,395.687,170.377,41.387,157.838
C08841=1037.960,203.520,395.662,170.380,41.388,157.838
C08842=1037.966,203.770,395.637,170.383,41.388,157.838
C08843=1037.972,204.006,395.613,170.387,41.388,157.839
C08844=1037.977,204.243,395.590,170.389,41.389,157.839
C08845=1037.983,204.479,395.565,170.392,41.390,157.839
C08846=1038.013,205.663,395.445,170.696,41.494,157.878
C08847=1038.021,205.981,395.412,170.699,41.496,157.879
C08848=1038.030,206.299,395.378,170.702,41.497,157.879
C08849=1038.039,206.617,395.345,170.705,41.499,157.880
C08850=1038.048,206.935,395.310,170.708,41.500,157.880
C08851=1038.054,207.183,395.284,170.710,41.501,157.880
C08852=1038.061,207.432,395.257,170.713,41.503,157.881
C08853=1038.067,207.680,395.231,170.715,41.504,157.881
C08854=1038.074,207.929,395.205,170.717,41.506,157.882
C08855=1038.081,208.178,395.178,170.719,41.507,157.882
C08856=1038.087,208.426,395.152,170.722,41.508,157.882
C08857=1038.094,208.675,395.125,170.724,41.509,157.883
C08858=1038.101,208.924,395.099,170.727,41.510,157.883
C08859=1038.108,209.171,395.072,170.729,41.512,157.884
C08860=1038.115,209.420,395.045,170.731,41.513,157.884
C08861=1038.120,209.668,395.018,170.734,41.514,157.885
C08862=1038.128,209.917,394.992,170.735,41.516,157.885
C08863=1038.135,210.166,394.966,170.738,41.517,157.885
C08864=1038.140,210.414,394.939,170.740,41.518,157.886
C08865=1038.148,210.662,394.912,170.743,41.519,157.886
C08866=1038.155,210.911,394.885,170.745,41.521,157.887
C08867=1038.161,211.159,394.859,170.748,41.522,157.887
C08868=1038.168,211.408,394.832,170.750,41.523,157.887
C08869=1038.175,211.657,394.805,170.753,41.524,157.888
C08870=1038.181,211.905,394.779,170.755,41.526,157.888
C08871=1038.187,212.154,394.752,170.756,41.527,157.889
C08872=1038.195,212.403,394.725,170.759,41.529,157.889
C08873=1038.201,212.650,394.698,170.761,41.530,157.889
C08874=1038.208,212.899,394.671,170.764,41.531,157.890
C08875=1038.214,213.148,394.644,170.766,41.532,157.890
C08876=1038.221,213.395,394.618,170.769,41.534,157.891
C08877=1038.227,213.645,394.591,170.771,41.535,157.891
C08878=1038.235,213.893,394.563,170.774,41.536,157.891
C08879=1038.241,214.141,394.537,170.776,41.537,157.892
C08880=1038.248,214.390,394.510,170.779,41.539,157.892
C08881=1038.254,214.638,394.483,170.780,41.540,157.893
C08882=1038.261,214.886,394.457,170.783,41.542,157.893
C08883=1038.267,215.135,394.430,170.785,41.543,157.893
C08884=1038.274,215.384,394.402,170.788,41.544,157.894
C08885=1038.281,215.633,394.375,170.790,41.545,157.894
C08886=1038.287,215.880,394.348,170.793,41.547,157.895
C08887=1038.294,216.129,394.322,170.795,41.548,157.895
C08888=1038.301,216.377,394.294,170.797,41.549,157.896
C08889=1038.308,216.626,394.267,170.800,41.550,157.896
C08890=1038.314,216.874,394.240,170.802,41.552,157.896
C08891=1038.321,217.123,394.214,170.805,41.553,157.897
C08892=1038.328,217.371,394.186,170.807,41.555,157.897
C08893=1038.334,217.620,394.159,170.810,41.556,157.898
C08894=1038.341,217.868,394.132,170.812,41.557,157.898
C08895=1038.347,218.117,394.105,170.815,41.558,157.898
C08896=1038.355,218.365,394.078,170.817,41.560,157.899
C08897=1038.361,218.614,394.051,170.820,41.561,157.899
C08898=1038.369,218.862,394.024,170.822,41.562,157.900
C08899=1038.374,219.110,393.997,170.824,41.563,157.900
C08900=1038.381,219.359,393.969,170.827,41.564,157.900
C08901=1038.388,219.608,393.943,170.829,41.566,157.901
C08902=1038.395,219.856,393.915,170.832,41.567,157.901
C08903=1038.404,220.180,393.880,170.835,41.569,157.902
C08904=1038.412,220.503,393.844,170.838,41.571,157.902
C08905=1038.421,220.827,393.808,170.842,41.572,157.903
C08906=1038.429,221.151,393.773,170.844,41.574,157.904
C08907=1038.436,221.399,393.745,170.847,41.575,157.904
C08908=1038.443,221.648,393.719,170.849,41.577,157.904
C08909=1038.450,221.896,393.691,170.852,41.578,157.905
C08910=1038.456,222.145,393.664,170.854,41.579,157.905
C08911=1038.462,222.392,393.636,170.857,41.580,157.906
C08912=1038.469,222.641,393.609,170.859,41.582,157.906
C08913=1038.475,222.890,393.581,170.862,41.584,157.907
C08914=1038.482,223.138,393.554,170.864,41.585,157.907
C08915=1038.490,223.386,393.527,170.867,41.586,157.907
C08916=1038.496,223.635,393.500,170.869,41.587,157.908
C08917=1038.503,223.884,393.472,170.872,41.589,157.908
C08918=1038.509,224.132,393.444,170.874,41.590,157.909
C08919=1038.515,224.380,393.417,170.877,41.591,157.909
C08920=1038.522,224.629,393.389,170.879,41.592,157.909
C08921=1038.529,224.877,393.362,170.882,41.594,157.910
C08922=1038.536,225.126,393.335,170.885,41.595,157.910
C08923=1038.542,225.374,393.307,170.887,41.596,157.911
C08924=1038.549,225.623,393.279,170.890,41.598,157.911
C08925=1038.556,225.871,393.252,170.892,41.599,157.912
C08926=1038.563,226.119,393.224,170.895,41.600,157.912
C08927=1038.569,226.367,393.197,170.897,41.601,157.912
C08928=1038.576,226.615,393.169,170.900,41.603,157.913
C08929=1038.583,226.864,393.142,170.902,41.604,157.913
C08930=1038.589,227.112,393.114,170.905,41.606,157.914
C08931=1038.596,227.361,393.086,170.907,41.606,157.914
C08932=1038.602,227.610,393.059,170.910,41.608,157.915
C08933=1038.609,227.858,393.031,170.912,41.609,157.915
C08934=1038.616,228.107,393.004,170.915,41.611,157.915
C08935=1038.623,228.355,392.976,170.918,41.611,157.916
C08936=1038.629,228.604,392.948,170.921,41.613,157.916
C08937=1038.636,228.852,392.921,170.923,41.615,157.917
C08938=1038.643,229.100,392.892,170.926,41.616,157.917
C08939=1038.650,229.348,392.864,170.928,41.617,157.918
C08940=1038.656,229.597,392.837,170.931,41.619,157.918
C08941=1038.663,229.845,392.809,170.933,41.620,157.918
C08942=1038.670,230.094,392.781,170.936,41.621,157.919
C08943=1038.676,230.342,392.753,170.938,41.622,157.919
C08944=1038.683,230.590,392.726,170.941,41.624,157.920
C08945=1038.690,230.839,392.698,170.943,41.626,157.920
C08946=1038.696,231.087,392.670,170.947,41.626,157.921
C08947=1038.703,231.335,392.641,170.949,41.628,157.921
C08948=1038.709,231.584,392.613,170.952,41.630,157.922
C08949=1038.716,231.832,392.586,170.954,41.630,157.922
C08950=1038.723,232.081,392.558,170.957,41.632,157.922
C08951=1038.729,232.329,392.530,170.959,41.633,157.923
C08952=1038.736,232.577,392.502,170.962,41.635,157.923
C08953=1038.742,232.826,392.474,170.964,41.636,157.924
C08954=1038.749,233.074,392.446,170.967,41.638,157.924
C08955=1038.756,233.323,392.418,170.970,41.639,157.925
C08956=1038.763,233.570,392.390,170.973,41.640,157.925
C08957=1038.769,233.819,392.361,170.975,41.642,157.926
C08958=1038.775,234.068,392.334,170.978,41.643,157.926
C08959=1038.785,234.450,392.290,170.981,41.645,157.927
C08960=1038.796,234.832,392.247,170.986,41.647,157.927
C08961=1038.806,235.214,392.203,170.990,41.649,157.928
C08962=1038.816,235.597,392.160,170.994,41.652,157.929
C08963=1038.823,235.846,392.132,170.996,41.652,157.929
C08964=1038.830,236.094,392.104,171.000,41.654,157.930
C08965=1038.836,236.342,392.075,171.002,41.656,157.930
C08966=1038.843,236.590,392.047,171.005,41.656,157.930
C08967=1038.849,236.839,392.019,171.007,41.658,157.931
C08968=1038.856,237.087,391.991,171.010,41.660,157.931
C08969=1038.862,237.335,391.962,171.012,41.661,157.932
C08970=1038.869,237.584,391.935,171.016,41.662,157.932
C08971=1038.875,237.799,391.910,171.018,41.663,157.933
C08972=1038.882,238.014,391.885,171.020,41.665,157.933
C08973=1038.886,238.229,391.861,171.022,41.666,157.933
C08974=1038.892,238.445,391.837,171.025,41.667,157.934
C08975=1038.898,238.659,391.812,171.027,41.668,157.934
C08976=1038.904,238.875,391.787,171.029,41.669,157.935
C08977=1038.910,239.091,391.763,171.032,41.670,157.935
C08978=1038.916,239.305,391.738,171.034,41.672,157.935
C08979=1038.923,239.554,391.710,171.037,41.673,157.936
C08980=1038.929,239.802,391.681,171.039,41.674,157.936
C08981=1038.936,240.050,391.653,171.043,41.676,157.937
C08982=1038.942,240.299,391.624,171.045,41.677,157.937
C08983=1038.949,240.546,391.596,171.048,41.678,157.938
C08984=1038.956,240.795,391.568,171.050,41.680,157.938
C08985=1038.963,241.044,391.539,171.054,41.681,157.938
C08986=1038.969,241.292,391.511,171.056,41.682,157.939
C08987=1038.976,241.540,391.482,171.059,41.684,157.939
C08988=1038.983,241.788,391.453,171.062,41.685,157.940
C08989=1038.989,242.036,391.424,171.064,41.686,157.940
C08990=1038.995,242.285,391.396,171.067,41.688,157.941
C08991=1039.002,242.534,391.367,171.070,41.689,157.941
C08992=1039.009,242.782,391.338,171.073,41.691,157.942
C08993=1039.016,243.029,391.310,171.075,41.693,157.942
C08994=1039.021,243.278,391.281,171.079,41.693,157.943
C08995=1039.028,243.526,391.253,171.081,41.695,157.943
C08996=1039.035,243.774,391.224,171.084,41.697,157.944
C08997=1039.042,244.023,391.194,171.086,41.698,157.944
C08998=1039.049,244.271,391.166,171.090,41.700,157.945
C08999=1039.054,244.520,391.138,171.092,41.700,157.945
C09000=1039.061,244.767,391.109,171.095,41.702,157.946
C09001=1039.068,245.016,391.080,171.097,41.704,157.946
C09002=1039.075,245.264,391.051,171.101,41.705,157.947
C09003=1039.081,245.513,391.022,171.104,41.707,157.947
C09004=1039.088,245.760,390.993,171.106,41.708,157.948
C09005=1039.094,246.008,390.964,171.109,41.710,157.948
C09006=1039.101,246.257,390.935,171.112,41.711,157.948
C09007=1039.107,246.505,390.906,171.115,41.712,157.949
C09008=1039.113,246.754,390.877,171.117,41.714,157.949
C09009=1039.120,247.002,390.848,171.120,41.715,157.950
C09010=1039.127,247.249,390.819,171.123,41.717,157.950
C09011=1039.133,247.498,390.790,171.126,41.718,157.951
C09012=1039.140,247.746,390.761,171.128,41.720,157.951
C09013=1039.146,247.995,390.732,171.132,41.721,157.952
C09014=1039.152,248.243,390.703,171.135,41.723,157.952
C09015=1039.161,248.553,390.666,171.138,41.724,157.953
C09016=1039.169,248.864,390.630,171.142,41.726,157.954
C09017=1039.177,249.175,390.594,171.145,41.729,157.954
C09018=1039.185,249.484,390.557,171.148,41.730,157.955
C09019=1039.192,249.733,390.528,171.152,41.731,157.955
C09020=1039.199,249.981,390.499,171.154,41.733,157.956
C09021=1039.205,250.230,390.470,171.157,41.735,157.956
C09022=1039.211,250.477,390.440,171.161,41.736,157.957
C09023=1039.218,250.726,390.411,171.163,41.738,157.957
C09024=1039.225,250.974,390.382,171.166,41.739,157.958
C09025=1039.231,251.222,390.353,171.169,41.741,157.958
C09026=1039.238,251.471,390.324,171.172,41.742,157.959
C09027=1039.245,251.719,390.295,171.174,41.743,157.959
C09028=1039.252,251.967,390.265,171.178,41.745,157.960
C09029=1039.258,252.215,390.236,171.180,41.746,157.960
C09030=1039.264,252.463,390.207,171.183,41.748,157.961
C09031=1039.271,252.712,390.177,171.187,41.749,157.961
C09032=1039.278,252.959,390.148,171.189,41.751,157.962
C09033=1039.285,253.207,390.119,171.192,41.752,157.962
C09034=1039.291,253.456,390.090,171.195,41.754,157.963
C09035=1039.298,253.704,390.060,171.198,41.755,157.963
C09036=1039.305,253.953,390.030,171.201,41.757,157.964
C09037=1039.311,254.201,390.001,171.204,41.758,157.964
C09038=1039.317,254.449,389.972,171.206,41.759,157.965
C09039=1039.324,254.697,389.942,171.210,41.761,157.965
C09040=1039.331,254.945,389.913,171.213,41.762,157.966
C09041=1039.339,255.193,389.884,171.215,41.764,157.966
C09042=1039.345,255.441,389.855,171.219,41.765,157.967
C09043=1039.352,255.690,389.825,171.221,41.767,157.967
C09044=1039.358,255.938,389.796,171.225,41.768,157.968
C09045=1039.365,256.186,389.766,171.227,41.770,157.968
C09046=1039.372,256.434,389.736,171.231,41.771,157.969
C09047=1039.379,256.683,389.707,171.234,41.773,157.969
C09048=1039.385,256.931,389.678,171.236,41.774,157.970
C09049=1039.392,257.179,389.648,171.240,41.775,157.970
C09050=1039.398,257.427,389.619,171.242,41.777,157.970
C09051=1039.405,257.676,389.589,171.246,41.778,157.971
C09052=1039.412,257.923,389.560,171.248,41.780,157.971
C09053=1039.419,258.172,389.530,171.252,41.781,157.972
C09054=1039.426,258.420,389.501,171.254,41.783,157.973
C09055=1039.433,258.668,389.471,171.258,41.784,157.973
C09056=1039.439,258.916,389.442,171.261,41.786,157.974
C09057=1039.446,259.164,389.412,171.263,41.787,157.974
C09058=1039.453,259.412,389.383,171.267,41.789,157.975
C09059=1039.460,259.661,389.353,171.269,41.790,157.975
C09060=1039.467,259.909,389.322,171.273,41.792,157.976
C09061=1039.473,260.157,389.293,171.275,41.793,157.976
C09062=1039.480,260.405,389.263,171.279,41.795,157.977
C09063=1039.487,260.653,389.234,171.282,41.796,157.977
C09064=1039.494,260.901,389.204,171.285,41.797,157.977
C09065=1039.502,261.149,389.175,171.288,41.798,157.978
C09066=1039.508,261.398,389.146,171.291,41.800,157.978
C09067=1039.515,261.646,389.115,171.294,41.801,157.979
C09068=1039.522,261.893,389.086,171.297,41.803,157.980
C09069=1039.528,262.142,389.056,171.300,41.804,157.980
C09070=1039.534,262.390,389.026,171.304,41.806,157.981
C09071=1039.543,262.699,388.988,171.307,41.808,157.981
C09072=1039.552,263.008,388.951,171.311,41.810,157.982
C09073=1039.559,263.317,388.914,171.315,41.812,157.983
C09074=1039.568,263.626,388.876,171.319,41.814,157.983
C09075=1039.574,263.874,388.846,171.322,41.815,157.984
C09076=1039.581,264.122,388.816,171.325,41.817,157.984
C09077=1039.587,264.371,388.786,171.328,41.818,157.985
C09078=1039.594,264.619,388.756,171.331,41.820,157.985
C09079=1039.601,264.867,388.726,171.335,41.822,157.986
C09080=1039.608,265.115,388.695,171.337,41.823,157.986
C09081=1039.614,265.363,388.665,171.341,41.825,157.987
C09082=1039.621,265.611,388.635,171.343,41.826,157.987
C09083=1039.628,265.858,388.606,171.347,41.828,157.988
C09084=1039.634,266.107,388.575,171.350,41.829,157.988
C09085=1039.641,266.355,388.545,171.353,41.831,157.989
C09086=1039.648,266.603,388.515,171.356,41.833,157.990
C09087=1039.654,266.851,388.484,171.360,41.834,157.990
C09088=1039.662,267.099,388.454,171.363,41.836,157.991
C09089=1039.668,267.347,388.424,171.366,41.837,157.991
C09090=1039.675,267.596,388.394,171.369,41.839,157.992
C09091=1039.682,267.844,388.364,171.372,41.841,157.992
C09092=1039.688,268.092,388.332,171.376,41.842,157.993
C09093=1039.695,268.339,388.302,171.378,41.844,157.993
C09094=1039.701,268.588,388.272,171.382,41.845,157.994
C09095=1039.709,268.836,388.242,171.384,41.847,157.994
C09096=1039.714,269.084,388.211,171.388,41.849,157.995
C09097=1039.721,269.332,388.181,171.391,41.850,157.996
C09098=1039.728,269.580,388.150,171.394,41.852,157.996
C09099=1039.735,269.827,388.120,171.398,41.853,157.997
C09100=1039.741,270.076,388.089,171.401,41.855,157.997
C09101=1039.748,270.324,388.059,171.404,41.857,157.998
C09102=1039.755,270.573,388.028,171.407,41.858,157.998
C09103=1039.762,270.819,387.998,171.410,41.860,157.999
C09104=1039.768,271.068,387.967,171.414,41.862,158.000
C09105=1039.775,271.316,387.937,171.417,41.863,158.000
